LIN {X 0,Y 255.137,Z 1284.988,A -85,B 0,C 180,E1 17189.999,E2 17189.999} C_VEL
LIN {X 0,Y 254.468,Z 1282.963,A -85,B 0,C 180,E1 17196.81,E2 17196.81} C_VEL
LIN {X 0,Y 254.384,Z 1277.292,A -85,B 0,C 180,E1 17203.725,E2 17203.725} C_VEL
LIN {X 0,Y 256.072,Z 1266.53,A -85,B 0,C 180,E1 17211.61,E2 17211.61} C_VEL
LIN {X 0,Y 262.116,Z 1248.09,A -85,B 0,C 180,E1 17220.546,E2 17220.546} C_VEL
LIN {X 0,Y 272.188,Z 1225.017,A -85,B 0,C 180,E1 17228.249,E2 17228.249} C_VEL
LIN {X 0,Y 284.902,Z 1198.098,A -85,B 0,C 180,E1 17234.56,E2 17234.56} C_VEL
LIN {X 0,Y 299.3,Z 1166.688,A -85,B 0,C 180,E1 17239.69,E2 17239.69} C_VEL
LIN {X 0,Y 313.161,Z 1132.639,A -85,B 0,C 180,E1 17243.514,E2 17243.514} C_VEL
LIN {X 0,Y 320.37,Z 1111.086,A -85,B 0,C 180,E1 17245.369,E2 17245.369} C_VEL
LIN {X 0,Y 312.607,Z 1086.253,A -85,B 0,C 180,E1 17250.782,E2 17250.782} C_VEL
LIN {X 0,Y 302.724,Z 1063.673,A -85,B 0,C 180,E1 17257.275,E2 17257.275} C_VEL
LIN {X 0,Y 294.391,Z 1048.168,A -85,B 0,C 180,E1 17263.626,E2 17263.626} C_VEL
LIN {X 0,Y 291.709,Z 1044.139,A -85,B 0,C 180,E1 17266.011,E2 17266.011} C_VEL
LIN {X 0,Y 289.339,Z 1043.796,A -85,B 0,C 180,E1 17267.674,E2 17267.674} C_VEL
LIN {X 0,Y 285.403,Z 1045.605,A -85,B 0,C 180,E1 17270.235,E2 17270.235} C_VEL
LIN {X 0,Y 285.166,Z 1045.322,A -85,B 0,C 180,E1 17270.526,E2 17270.526} C_VEL
LIN {X 0,Y 284.224,Z 1042.423,A -85,B 0,C 180,E1 17272.373,E2 17272.373} C_VEL
LIN {X 0,Y 280.854,Z 1038.34,A -85,B 0,C 180,E1 17280,E2 17280} C_VEL
LIN {X 0,Y 280.283,Z 1039.511,A -85,B 0,C 180,E1 17286.181,E2 17286.181} C_VEL
LIN {X 0,Y 281.282,Z 1041.764,A -85,B 0,C 180,E1 17290.897,E2 17290.897} C_VEL
LIN {X 0,Y 284.187,Z 1051.363,A -85,B 0,C 180,E1 17298.577,E2 17298.577} C_VEL
LIN {X 0,Y 287.728,Z 1062.486,A -85,B 0,C 180,E1 17304.806,E2 17304.806} C_VEL
LIN {X 0,Y 291.72,Z 1079.881,A -85,B 0,C 180,E1 17312.089,E2 17312.089} C_VEL
LIN {X 0,Y 294.002,Z 1097.791,A -85,B 0,C 180,E1 17318.393,E2 17318.393} C_VEL
LIN {X 0,Y 294.147,Z 1115.354,A -85,B 0,C 180,E1 17324.094,E2 17324.094} C_VEL
LIN {X 0,Y 280.403,Z 1140.437,A -85,B 0,C 180,E1 17329.776,E2 17329.776} C_VEL
LIN {X 0,Y 267.571,Z 1161.591,A -85,B 0,C 180,E1 17336.74,E2 17336.74} C_VEL
LIN {X 0,Y 257.328,Z 1177.923,A -85,B 0,C 180,E1 17344.841,E2 17344.841} C_VEL
LIN {X 0,Y 251.436,Z 1187.855,A -85,B 0,C 180,E1 17352.539,E2 17352.539} C_VEL
LIN {X 0,Y 248.589,Z 1193.315,A -85,B 0,C 180,E1 17359.509,E2 17359.509} C_VEL
LIN {X 0,Y 247.507,Z 1195.971,A -85,B 0,C 180,E1 17366.506,E2 17366.506} C_VEL
LIN {X 0,Y 247.516,Z 1195.938,A -85,B 0,C 180,E1 17373.497,E2 17373.497} C_VEL
LIN {X 0,Y 249.137,Z 1192.204,A -85,B 0,C 180,E1 17382.24,E2 17382.24} C_VEL
LIN {X 0,Y 254.389,Z 1182.789,A -85,B 0,C 180,E1 17391.718,E2 17391.718} C_VEL
LIN {X 0,Y 263.096,Z 1168.574,A -85,B 0,C 180,E1 17400.125,E2 17400.125} C_VEL
LIN {X 0,Y 275.237,Z 1149.075,A -85,B 0,C 180,E1 17407.586,E2 17407.586} C_VEL
LIN {X 0,Y 288.938,Z 1125.242,A -85,B 0,C 180,E1 17413.775,E2 17413.775} C_VEL
LIN {X 0,Y 294.085,Z 1114.963,A -85,B 0,C 180,E1 17415.921,E2 17415.921} C_VEL
LIN {X 0,Y 293.829,Z 1096.412,A -85,B 0,C 180,E1 17421.957,E2 17421.957} C_VEL
LIN {X 0,Y 291.448,Z 1078.298,A -85,B 0,C 180,E1 17428.357,E2 17428.357} C_VEL
LIN {X 0,Y 287.609,Z 1062.12,A -85,B 0,C 180,E1 17435.183,E2 17435.183} C_VEL
LIN {X 0,Y 283.183,Z 1048.498,A -85,B 0,C 180,E1 17443.118,E2 17443.118} C_VEL
LIN {X 0,Y 280.59,Z 1040.614,A -85,B 0,C 180,E1 17450.716,E2 17450.716} C_VEL
LIN {X 0,Y 280.229,Z 1037.979,A -85,B 0,C 180,E1 17456.913,E2 17456.913} C_VEL
LIN {X 0,Y 280.753,Z 1037.906,A -85,B 0,C 180,E1 17460,E2 17460} C_VEL
LIN {X 0,Y 284.152,Z 1041.989,A -85,B 0,C 180,E1 17467.629,E2 17467.629} C_VEL
LIN {X 0,Y 290.868,Z 1054.58,A -85,B 0,C 180,E1 17475.805,E2 17475.805} C_VEL
LIN {X 0,Y 299.294,Z 1071.309,A -85,B 0,C 180,E1 17482.717,E2 17482.717} C_VEL
LIN {X 0,Y 307.569,Z 1091.151,A -85,B 0,C 180,E1 17488.576,E2 17488.576} C_VEL
LIN {X 0,Y 314.317,Z 1114.372,A -85,B 0,C 180,E1 17493.824,E2 17493.824} C_VEL
LIN {X 0,Y 300.167,Z 1151.228,A -85,B 0,C 180,E1 17497.349,E2 17497.349} C_VEL
LIN {X 0,Y 285.171,Z 1183.85,A -85,B 0,C 180,E1 17501.908,E2 17501.908} C_VEL
LIN {X 0,Y 270.591,Z 1213.505,A -85,B 0,C 180,E1 17507.992,E2 17507.992} C_VEL
LIN {X 0,Y 258.739,Z 1238.273,A -85,B 0,C 180,E1 17515.343,E2 17515.343} C_VEL
LIN {X 0,Y 250.401,Z 1258.673,A -85,B 0,C 180,E1 17524.093,E2 17524.093} C_VEL
LIN {X 0,Y 246.852,Z 1272.762,A -85,B 0,C 180,E1 17533.119,E2 17533.119} C_VEL
LIN {X 0,Y 246.557,Z 1280.502,A -85,B 0,C 180,E1 17541.197,E2 17541.197} C_VEL
LIN {X 0,Y 246.904,Z 1283.038,A -85,B 0,C 180,E1 17546.495,E2 17546.495} C_VEL
LIN {X 0,Y 247.367,Z 1283.617,A -85,B 0,C 180,E1 17549.999,E2 17549.999} C_VEL
LIN {X 0,Y 246.653,Z 1281.574,A -85,B 0,C 180,E1 17557.027,E2 17557.027} C_VEL
LIN {X 0,Y 246.583,Z 1275.874,A -85,B 0,C 180,E1 17564.168,E2 17564.168} C_VEL
LIN {X 0,Y 248.469,Z 1265.084,A -85,B 0,C 180,E1 17572.306,E2 17572.306} C_VEL
LIN {X 0,Y 254.378,Z 1248.105,A -85,B 0,C 180,E1 17580.899,E2 17580.899} C_VEL
LIN {X 0,Y 264.784,Z 1225.469,A -85,B 0,C 180,E1 17588.82,E2 17588.82} C_VEL
LIN {X 0,Y 278.173,Z 1198.463,A -85,B 0,C 180,E1 17595.396,E2 17595.396} C_VEL
LIN {X 0,Y 293.472,Z 1166.431,A -85,B 0,C 180,E1 17600.758,E2 17600.758} C_VEL
LIN {X 0,Y 307.806,Z 1132.751,A -85,B 0,C 180,E1 17604.588,E2 17604.588} C_VEL
LIN {X 0,Y 314.425,Z 1114.35,A -85,B 0,C 180,E1 17606.188,E2 17606.188} C_VEL
LIN {X 0,Y 307.121,Z 1089.98,A -85,B 0,C 180,E1 17611.779,E2 17611.779} C_VEL
LIN {X 0,Y 298.39,Z 1069.256,A -85,B 0,C 180,E1 17618.051,E2 17618.051} C_VEL
LIN {X 0,Y 290.985,Z 1054.781,A -85,B 0,C 180,E1 17624.202,E2 17624.202} C_VEL
LIN {X 0,Y 287.467,Z 1048.317,A -85,B 0,C 180,E1 17627.88,E2 17627.88} C_VEL
LIN {X 0,Y 285.166,Z 1045.322,A -85,B 0,C 180,E1 17630.526,E2 17630.526} C_VEL
LIN {X 0,Y 282.691,Z 1044.878,A -85,B 0,C 180,E1 17633.12,E2 17633.12} C_VEL
LIN {X 0,Y 278.853,Z 1047.015,A -85,B 0,C 180,E1 17637.566,E2 17637.566} C_VEL
LIN {X 0,Y 277.646,Z 1045.811,A -85,B 0,C 180,E1 17643.115,E2 17643.115} C_VEL
LIN {X 0,Y 278.291,Z 1049.367,A -85,B 0,C 180,E1 17651.015,E2 17651.015} C_VEL
LIN {X 0,Y 280.713,Z 1058.959,A -85,B 0,C 180,E1 17658.816,E2 17658.816} C_VEL
LIN {X 0,Y 284.069,Z 1071.905,A -85,B 0,C 180,E1 17665.873,E2 17665.873} C_VEL
LIN {X 0,Y 286.988,Z 1088.241,A -85,B 0,C 180,E1 17672.725,E2 17672.725} C_VEL
LIN {X 0,Y 288.302,Z 1105.417,A -85,B 0,C 180,E1 17678.908,E2 17678.908} C_VEL
LIN {X 0,Y 287.43,Z 1119.484,A -85,B 0,C 180,E1 17683.545,E2 17683.545} C_VEL
LIN {X 0,Y 272.089,Z 1145.854,A -85,B 0,C 180,E1 17689.856,E2 17689.856} C_VEL
LIN {X 0,Y 258.657,Z 1166.631,A -85,B 0,C 180,E1 17697.342,E2 17697.342} C_VEL
LIN {X 0,Y 248.492,Z 1182.013,A -85,B 0,C 180,E1 17705.895,E2 17705.895} C_VEL
LIN {X 0,Y 242.157,Z 1192.333,A -85,B 0,C 180,E1 17715.567,E2 17715.567} C_VEL
LIN {X 0,Y 240.061,Z 1196.366,A -85,B 0,C 180,E1 17722.779,E2 17722.779} C_VEL
LIN {X 0,Y 239.805,Z 1197.644,A -85,B 0,C 180,E1 17730.001,E2 17730.001} C_VEL
LIN {X 0,Y 240.054,Z 1196.316,A -85,B 0,C 180,E1 17737.224,E2 17737.224} C_VEL
LIN {X 0,Y 242.888,Z 1191.132,A -85,B 0,C 180,E1 17745.877,E2 17745.877} C_VEL
LIN {X 0,Y 249.513,Z 1180.492,A -85,B 0,C 180,E1 17755.047,E2 17755.047} C_VEL
LIN {X 0,Y 259.981,Z 1164.513,A -85,B 0,C 180,E1 17763.465,E2 17763.465} C_VEL
LIN {X 0,Y 273.017,Z 1144.178,A -85,B 0,C 180,E1 17770.501,E2 17770.501} C_VEL
LIN {X 0,Y 287.455,Z 1119.187,A -85,B 0,C 180,E1 17776.414,E2 17776.414} C_VEL
LIN {X 0,Y 288.073,Z 1103.066,A -85,B 0,C 180,E1 17781.791,E2 17781.791} C_VEL
LIN {X 0,Y 286.553,Z 1085.286,A -85,B 0,C 180,E1 17788.225,E2 17788.225} C_VEL
LIN {X 0,Y 283.263,Z 1068.551,A -85,B 0,C 180,E1 17795.523,E2 17795.523} C_VEL
LIN {X 0,Y 279.675,Z 1055.247,A -85,B 0,C 180,E1 17803.552,E2 17803.552} C_VEL
LIN {X 0,Y 277.738,Z 1048.039,A -85,B 0,C 180,E1 17810.62,E2 17810.62} C_VEL
LIN {X 0,Y 277.527,Z 1045.448,A -85,B 0,C 180,E1 17816.883,E2 17816.883} C_VEL
LIN {X 0,Y 278.18,Z 1045.394,A -85,B 0,C 180,E1 17820,E2 17820} C_VEL
LIN {X 0,Y 281.517,Z 1049.856,A -85,B 0,C 180,E1 17827.701,E2 17827.701} C_VEL
LIN {X 0,Y 287.342,Z 1061.146,A -85,B 0,C 180,E1 17835.223,E2 17835.223} C_VEL
LIN {X 0,Y 295.025,Z 1076.971,A -85,B 0,C 180,E1 17842.018,E2 17842.018} C_VEL
LIN {X 0,Y 302.864,Z 1097.215,A -85,B 0,C 180,E1 17848.183,E2 17848.183} C_VEL
LIN {X 0,Y 308.379,Z 1117.716,A -85,B 0,C 180,E1 17853.017,E2 17853.017} C_VEL
LIN {X 0,Y 294.309,Z 1151.941,A -85,B 0,C 180,E1 17856.342,E2 17856.342} C_VEL
LIN {X 0,Y 278.69,Z 1184.433,A -85,B 0,C 180,E1 17861.002,E2 17861.002} C_VEL
LIN {X 0,Y 263.917,Z 1213.139,A -85,B 0,C 180,E1 17867.067,E2 17867.067} C_VEL
LIN {X 0,Y 251.35,Z 1237.996,A -85,B 0,C 180,E1 17874.7,E2 17874.7} C_VEL
LIN {X 0,Y 243.009,Z 1257.212,A -85,B 0,C 180,E1 17883.242,E2 17883.242} C_VEL
LIN {X 0,Y 239.101,Z 1271.33,A -85,B 0,C 180,E1 17892.554,E2 17892.554} C_VEL
LIN {X 0,Y 238.711,Z 1279.1,A -85,B 0,C 180,E1 17900.906,E2 17900.906} C_VEL
LIN {X 0,Y 239.099,Z 1281.658,A -85,B 0,C 180,E1 17906.38,E2 17906.38} C_VEL
LIN {X 0,Y 239.571,Z 1282.241,A -85,B 0,C 180,E1 17909.999,E2 17909.999} C_VEL
LIN {X 0,Y 238.828,Z 1280.182,A -85,B 0,C 180,E1 17917.258,E2 17917.258} C_VEL
LIN {X 0,Y 238.788,Z 1274.454,A -85,B 0,C 180,E1 17924.641,E2 17924.641} C_VEL
LIN {X 0,Y 241.327,Z 1262.214,A -85,B 0,C 180,E1 17933.91,E2 17933.91} C_VEL
LIN {X 0,Y 248.706,Z 1243.691,A -85,B 0,C 180,E1 17943.096,E2 17943.096} C_VEL
LIN {X 0,Y 260.58,Z 1219.799,A -85,B 0,C 180,E1 17951.167,E2 17951.167} C_VEL
LIN {X 0,Y 275.272,Z 1191.427,A -85,B 0,C 180,E1 17957.735,E2 17957.735} C_VEL
LIN {X 0,Y 291.413,Z 1158.364,A -85,B 0,C 180,E1 17962.918,E2 17962.918} C_VEL
LIN {X 0,Y 306.908,Z 1121.702,A -85,B 0,C 180,E1 17966.704,E2 17966.704} C_VEL
LIN {X 0,Y 308.352,Z 1117.832,A -85,B 0,C 180,E1 17967.005,E2 17967.005} C_VEL
LIN {X 0,Y 302.38,Z 1095.769,A -85,B 0,C 180,E1 17972.257,E2 17972.257} C_VEL
LIN {X 0,Y 294.431,Z 1075.586,A -85,B 0,C 180,E1 17978.548,E2 17978.548} C_VEL
LIN {X 0,Y 287.451,Z 1061.347,A -85,B 0,C 180,E1 17984.783,E2 17984.783} C_VEL
LIN {X 0,Y 281.577,Z 1050.332,A -85,B 0,C 180,E1 17992.301,E2 17992.301} C_VEL
LIN {X 0,Y 278.853,Z 1047.015,A -85,B 0,C 180,E1 17997.566,E2 17997.566} C_VEL
LIN {X 0,Y 277.184,Z 1048.421,A -85,B 0,C 180,E1 18000.225,E2 18000.225} C_VEL
LIN {X 0,Y 274.51,Z 1053.721,A -85,B 0,C 180,E1 18004.671,E2 18004.671} C_VEL
LIN {X 0,Y 275.027,Z 1056.889,A -85,B 0,C 180,E1 18011.148,E2 18011.148} C_VEL
LIN {X 0,Y 277.086,Z 1066.535,A -85,B 0,C 180,E1 18019.071,E2 18019.071} C_VEL
LIN {X 0,Y 279.809,Z 1079.929,A -85,B 0,C 180,E1 18026.417,E2 18026.417} C_VEL
LIN {X 0,Y 281.865,Z 1096.426,A -85,B 0,C 180,E1 18033.396,E2 18033.396} C_VEL
LIN {X 0,Y 282.223,Z 1115.213,A -85,B 0,C 180,E1 18040.301,E2 18040.301} C_VEL
LIN {X 0,Y 281.309,Z 1122.317,A -85,B 0,C 180,E1 18042.676,E2 18042.676} C_VEL
LIN {X 0,Y 265.31,Z 1148.466,A -85,B 0,C 180,E1 18049.151,E2 18049.151} C_VEL
LIN {X 0,Y 252.074,Z 1168.017,A -85,B 0,C 180,E1 18056.377,E2 18056.377} C_VEL
LIN {X 0,Y 241.347,Z 1183.397,A -85,B 0,C 180,E1 18065.134,E2 18065.134} C_VEL
LIN {X 0,Y 234.584,Z 1193.714,A -85,B 0,C 180,E1 18075.091,E2 18075.091} C_VEL
LIN {X 0,Y 232.329,Z 1197.741,A -85,B 0,C 180,E1 18082.537,E2 18082.537} C_VEL
LIN {X 0,Y 232.043,Z 1199.014,A -85,B 0,C 180,E1 18090.001,E2 18090.001} C_VEL
LIN {X 0,Y 232.32,Z 1197.693,A -85,B 0,C 180,E1 18097.466,E2 18097.466} C_VEL
LIN {X 0,Y 235.525,Z 1192.196,A -85,B 0,C 180,E1 18106.757,E2 18106.757} C_VEL
LIN {X 0,Y 242.427,Z 1181.878,A -85,B 0,C 180,E1 18115.833,E2 18115.833} C_VEL
LIN {X 0,Y 253.473,Z 1165.899,A -85,B 0,C 180,E1 18124.443,E2 18124.443} C_VEL
LIN {X 0,Y 267.117,Z 1145.561,A -85,B 0,C 180,E1 18131.591,E2 18131.591} C_VEL
LIN {X 0,Y 281.614,Z 1120.703,A -85,B 0,C 180,E1 18137.677,E2 18137.677} C_VEL
LIN {X 0,Y 282.138,Z 1101.835,A -85,B 0,C 180,E1 18144.395,E2 18144.395} C_VEL
LIN {X 0,Y 280.573,Z 1085.149,A -85,B 0,C 180,E1 18151.051,E2 18151.051} C_VEL
LIN {X 0,Y 277.834,Z 1070.385,A -85,B 0,C 180,E1 18158.361,E2 18158.361} C_VEL
LIN {X 0,Y 275.38,Z 1059.996,A -85,B 0,C 180,E1 18165.725,E2 18165.725} C_VEL
LIN {X 0,Y 274.363,Z 1054.762,A -85,B 0,C 180,E1 18171.902,E2 18171.902} C_VEL
LIN {X 0,Y 275.302,Z 1052.79,A -85,B 0,C 180,E1 18180,E2 18180} C_VEL
LIN {X 0,Y 278.589,Z 1057.631,A -85,B 0,C 180,E1 18187.782,E2 18187.782} C_VEL
LIN {X 0,Y 284.37,Z 1069.061,A -85,B 0,C 180,E1 18195.386,E2 18195.386} C_VEL
LIN {X 0,Y 291.065,Z 1083.921,A -85,B 0,C 180,E1 18201.805,E2 18201.805} C_VEL
LIN {X 0,Y 298.159,Z 1103.61,A -85,B 0,C 180,E1 18207.913,E2 18207.913} C_VEL
LIN {X 0,Y 302.122,Z 1121.309,A -85,B 0,C 180,E1 18212.128,E2 18212.128} C_VEL
LIN {X 0,Y 286.317,Z 1157.309,A -85,B 0,C 180,E1 18215.852,E2 18215.852} C_VEL
LIN {X 0,Y 269.765,Z 1189.854,A -85,B 0,C 180,E1 18220.959,E2 18220.959} C_VEL
LIN {X 0,Y 254.209,Z 1218.36,A -85,B 0,C 180,E1 18227.613,E2 18227.613} C_VEL
LIN {X 0,Y 241.791,Z 1242.173,A -85,B 0,C 180,E1 18235.826,E2 18235.826} C_VEL
LIN {X 0,Y 233.939,Z 1260.374,A -85,B 0,C 180,E1 18245.048,E2 18245.048} C_VEL
LIN {X 0,Y 230.946,Z 1273.002,A -85,B 0,C 180,E1 18254.848,E2 18254.848} C_VEL
LIN {X 0,Y 231.033,Z 1278.783,A -85,B 0,C 180,E1 18262.493,E2 18262.493} C_VEL
LIN {X 0,Y 231.799,Z 1280.869,A -85,B 0,C 180,E1 18269.999,E2 18269.999} C_VEL
LIN {X 0,Y 231.004,Z 1278.791,A -85,B 0,C 180,E1 18277.506,E2 18277.506} C_VEL
LIN {X 0,Y 230.969,Z 1273.027,A -85,B 0,C 180,E1 18285.148,E2 18285.148} C_VEL
LIN {X 0,Y 233.955,Z 1260.411,A -85,B 0,C 180,E1 18294.947,E2 18294.947} C_VEL
LIN {X 0,Y 241.783,Z 1242.225,A -85,B 0,C 180,E1 18304.172,E2 18304.172} C_VEL
LIN {X 0,Y 254.331,Z 1218.322,A -85,B 0,C 180,E1 18312.41,E2 18312.41} C_VEL
LIN {X 0,Y 269.789,Z 1189.973,A -85,B 0,C 180,E1 18319.032,E2 18319.032} C_VEL
LIN {X 0,Y 286.198,Z 1157.626,A -85,B 0,C 180,E1 18324.132,E2 18324.132} C_VEL
LIN {X 0,Y 302.386,Z 1120.228,A -85,B 0,C 180,E1 18328.032,E2 18328.032} C_VEL
LIN {X 0,Y 296.511,Z 1098.509,A -85,B 0,C 180,E1 18333.558,E2 18333.558} C_VEL
LIN {X 0,Y 288.998,Z 1078.92,A -85,B 0,C 180,E1 18340.159,E2 18340.159} C_VEL
LIN {X 0,Y 282.367,Z 1065.494,A -85,B 0,C 180,E1 18346.873,E2 18346.873} C_VEL
LIN {X 0,Y 277.822,Z 1056.475,A -85,B 0,C 180,E1 18353.764,E2 18353.764} C_VEL
LIN {X 0,Y 275.395,Z 1053.192,A -85,B 0,C 180,E1 18360,E2 18360} C_VEL
LIN {X 0,Y 274.51,Z 1053.721,A -85,B 0,C 180,E1 18364.671,E2 18364.671} C_VEL
LIN {X 0,Y 273.488,Z 1056.922,A -85,B 0,C 180,E1 18367.32,E2 18367.32} C_VEL
LIN {X 0,Y 271.581,Z 1064.694,A -85,B 0,C 180,E1 18371.664,E2 18371.664} C_VEL
LIN {X 0,Y 273.152,Z 1074.035,A -85,B 0,C 180,E1 18379.357,E2 18379.357} C_VEL
LIN {X 0,Y 275.15,Z 1087.013,A -85,B 0,C 180,E1 18386.554,E2 18386.554} C_VEL
LIN {X 0,Y 276.433,Z 1104.04,A -85,B 0,C 180,E1 18393.918,E2 18393.918} C_VEL
LIN {X 0,Y 275.791,Z 1121.552,A -85,B 0,C 180,E1 18400.552,E2 18400.552} C_VEL
LIN {X 0,Y 274.354,Z 1126.477,A -85,B 0,C 180,E1 18402.065,E2 18402.065} C_VEL
LIN {X 0,Y 258.578,Z 1151.073,A -85,B 0,C 180,E1 18408.409,E2 18408.409} C_VEL
LIN {X 0,Y 244.227,Z 1171.179,A -85,B 0,C 180,E1 18416.216,E2 18416.216} C_VEL
LIN {X 0,Y 234.116,Z 1184.962,A -85,B 0,C 180,E1 18424.467,E2 18424.467} C_VEL
LIN {X 0,Y 227.041,Z 1195.093,A -85,B 0,C 180,E1 18434.583,E2 18434.583} C_VEL
LIN {X 0,Y 224.609,Z 1199.115,A -85,B 0,C 180,E1 18442.279,E2 18442.279} C_VEL
LIN {X 0,Y 224.263,Z 1200.387,A -85,B 0,C 180,E1 18450.001,E2 18450.001} C_VEL
LIN {X 0,Y 224.6,Z 1199.067,A -85,B 0,C 180,E1 18457.724,E2 18457.724} C_VEL
LIN {X 0,Y 228.04,Z 1193.576,A -85,B 0,C 180,E1 18467.326,E2 18467.326} C_VEL
LIN {X 0,Y 235.395,Z 1183.263,A -85,B 0,C 180,E1 18476.664,E2 18476.664} C_VEL
LIN {X 0,Y 247.049,Z 1167.284,A -85,B 0,C 180,E1 18485.471,E2 18485.471} C_VEL
LIN {X 0,Y 261.316,Z 1146.944,A -85,B 0,C 180,E1 18492.73,E2 18492.73} C_VEL
LIN {X 0,Y 275.285,Z 1124.783,A -85,B 0,C 180,E1 18498.19,E2 18498.19} C_VEL
LIN {X 0,Y 276.431,Z 1107.448,A -85,B 0,C 180,E1 18504.624,E2 18504.624} C_VEL
LIN {X 0,Y 275.643,Z 1091.63,A -85,B 0,C 180,E1 18511.157,E2 18511.157} C_VEL
LIN {X 0,Y 273.726,Z 1077.748,A -85,B 0,C 180,E1 18518.156,E2 18518.156} C_VEL
LIN {X 0,Y 271.83,Z 1067.361,A -85,B 0,C 180,E1 18525.535,E2 18525.535} C_VEL
LIN {X 0,Y 271.311,Z 1062.741,A -85,B 0,C 180,E1 18530.395,E2 18530.395} C_VEL
LIN {X 0,Y 271.765,Z 1060.081,A -85,B 0,C 180,E1 18538.175,E2 18538.175} C_VEL
LIN {X 0,Y 273.117,Z 1061.867,A -85,B 0,C 180,E1 18543.167,E2 18543.167} C_VEL
LIN {X 0,Y 275.552,Z 1065.297,A -85,B 0,C 180,E1 18547.869,E2 18547.869} C_VEL
LIN {X 0,Y 280.473,Z 1075.379,A -85,B 0,C 180,E1 18554.805,E2 18554.805} C_VEL
LIN {X 0,Y 286.994,Z 1090.804,A -85,B 0,C 180,E1 18561.595,E2 18561.595} C_VEL
LIN {X 0,Y 293.218,Z 1109.68,A -85,B 0,C 180,E1 18567.591,E2 18567.591} C_VEL
LIN {X 0,Y 296.304,Z 1123.552,A -85,B 0,C 180,E1 18571.117,E2 18571.117} C_VEL
LIN {X 0,Y 280.399,Z 1158.219,A -85,B 0,C 180,E1 18574.812,E2 18574.812} C_VEL
LIN {X 0,Y 264.396,Z 1188.386,A -85,B 0,C 180,E1 18579.599,E2 18579.599} C_VEL
LIN {X 0,Y 248.225,Z 1216.661,A -85,B 0,C 180,E1 18586.246,E2 18586.246} C_VEL
LIN {X 0,Y 234.908,Z 1240.693,A -85,B 0,C 180,E1 18594.678,E2 18594.678} C_VEL
LIN {X 0,Y 226.39,Z 1259.205,A -85,B 0,C 180,E1 18604.353,E2 18604.353} C_VEL
LIN {X 0,Y 223.163,Z 1271.576,A -85,B 0,C 180,E1 18614.306,E2 18614.306} C_VEL
LIN {X 0,Y 223.184,Z 1277.385,A -85,B 0,C 180,E1 18622.227,E2 18622.227} C_VEL
LIN {X 0,Y 224.004,Z 1279.494,A -85,B 0,C 180,E1 18629.999,E2 18629.999} C_VEL
LIN {X 0,Y 223.153,Z 1277.393,A -85,B 0,C 180,E1 18637.771,E2 18637.771} C_VEL
LIN {X 0,Y 223.44,Z 1269.868,A -85,B 0,C 180,E1 18647.48,E2 18647.48} C_VEL
LIN {X 0,Y 227.613,Z 1256.069,A -85,B 0,C 180,E1 18657.649,E2 18657.649} C_VEL
LIN {X 0,Y 237.411,Z 1236.13,A -85,B 0,C 180,E1 18667.229,E2 18667.229} C_VEL
LIN {X 0,Y 251.74,Z 1210.753,A -85,B 0,C 180,E1 18675.386,E2 18675.386} C_VEL
LIN {X 0,Y 267.656,Z 1182.671,A -85,B 0,C 180,E1 18681.466,E2 18681.466} C_VEL
LIN {X 0,Y 284.393,Z 1150.164,A -85,B 0,C 180,E1 18686.215,E2 18686.215} C_VEL
LIN {X 0,Y 296.348,Z 1123.596,A -85,B 0,C 180,E1 18688.903,E2 18688.903} C_VEL
LIN {X 0,Y 291.398,Z 1103.386,A -85,B 0,C 180,E1 18694.298,E2 18694.298} C_VEL
LIN {X 0,Y 284.559,Z 1084.411,A -85,B 0,C 180,E1 18700.967,E2 18700.967} C_VEL
LIN {X 0,Y 278.135,Z 1070.556,A -85,B 0,C 180,E1 18708.261,E2 18708.261} C_VEL
LIN {X 0,Y 274.861,Z 1063.925,A -85,B 0,C 180,E1 18713.696,E2 18713.696} C_VEL
LIN {X 0,Y 272.368,Z 1060.505,A -85,B 0,C 180,E1 18720,E2 18720} C_VEL
LIN {X 0,Y 271.244,Z 1061.555,A -85,B 0,C 180,E1 18726.388,E2 18726.388} C_VEL
LIN {X 0,Y 271.581,Z 1064.694,A -85,B 0,C 180,E1 18731.664,E2 18731.664} C_VEL
LIN {X 0,Y 270.77,Z 1069.677,A -85,B 0,C 180,E1 18734.225,E2 18734.225} C_VEL
LIN {X 0,Y 268.802,Z 1079.659,A -85,B 0,C 180,E1 18738.406,E2 18738.406} C_VEL
LIN {X 0,Y 270.16,Z 1091.867,A -85,B 0,C 180,E1 18745.643,E2 18745.643} C_VEL
LIN {X 0,Y 270.795,Z 1107.938,A -85,B 0,C 180,E1 18752.969,E2 18752.969} C_VEL
LIN {X 0,Y 269.763,Z 1124.431,A -85,B 0,C 180,E1 18759.545,E2 18759.545} C_VEL
LIN {X 0,Y 268.2,Z 1129.4,A -85,B 0,C 180,E1 18761.166,E2 18761.166} C_VEL
LIN {X 0,Y 251.888,Z 1153.681,A -85,B 0,C 180,E1 18767.628,E2 18767.628} C_VEL
LIN {X 0,Y 237.743,Z 1172.562,A -85,B 0,C 180,E1 18775.164,E2 18775.164} C_VEL
LIN {X 0,Y 226.498,Z 1187.063,A -85,B 0,C 180,E1 18784.183,E2 18784.183} C_VEL
LIN {X 0,Y 219.326,Z 1196.724,A -85,B 0,C 180,E1 18794.405,E2 18794.405} C_VEL
LIN {X 0,Y 216.886,Z 1200.491,A -85,B 0,C 180,E1 18802.003,E2 18802.003} C_VEL
LIN {X 0,Y 216.5,Z 1201.757,A -85,B 0,C 180,E1 18810.001,E2 18810.001} C_VEL
LIN {X 0,Y 216.876,Z 1200.444,A -85,B 0,C 180,E1 18818.001,E2 18818.001} C_VEL
LIN {X 0,Y 220.593,Z 1194.956,A -85,B 0,C 180,E1 18827.93,E2 18827.93} C_VEL
LIN {X 0,Y 228.407,Z 1184.65,A -85,B 0,C 180,E1 18837.548,E2 18837.548} C_VEL
LIN {X 0,Y 240.71,Z 1168.669,A -85,B 0,C 180,E1 18846.554,E2 18846.554} C_VEL
LIN {X 0,Y 255.612,Z 1148.33,A -85,B 0,C 180,E1 18853.923,E2 18853.923} C_VEL
LIN {X 0,Y 268.911,Z 1128.12,A -85,B 0,C 180,E1 18858.995,E2 18858.995} C_VEL
LIN {X 0,Y 270.721,Z 1110.985,A -85,B 0,C 180,E1 18865.629,E2 18865.629} C_VEL
LIN {X 0,Y 270.401,Z 1096.305,A -85,B 0,C 180,E1 18872.026,E2 18872.026} C_VEL
LIN {X 0,Y 269.027,Z 1082.387,A -85,B 0,C 180,E1 18879.548,E2 18879.548} C_VEL
LIN {X 0,Y 267.828,Z 1073.013,A -85,B 0,C 180,E1 18886.976,E2 18886.976} C_VEL
LIN {X 0,Y 267.633,Z 1068.742,A -85,B 0,C 180,E1 18892.996,E2 18892.996} C_VEL
LIN {X 0,Y 269.091,Z 1067.35,A -85,B 0,C 180,E1 18900,E2 18900} C_VEL
LIN {X 0,Y 272.261,Z 1072.811,A -85,B 0,C 180,E1 18907.964,E2 18907.964} C_VEL
LIN {X 0,Y 276.872,Z 1082.542,A -85,B 0,C 180,E1 18914.68,E2 18914.68} C_VEL
LIN {X 0,Y 282.86,Z 1097.905,A -85,B 0,C 180,E1 18921.516,E2 18921.516} C_VEL
LIN {X 0,Y 288.421,Z 1116.605,A -85,B 0,C 180,E1 18927.526,E2 18927.526} C_VEL
LIN {X 0,Y 290.028,Z 1127.06,A -85,B 0,C 180,E1 18930.183,E2 18930.183} C_VEL
LIN {X 0,Y 273.255,Z 1161.673,A -85,B 0,C 180,E1 18934.068,E2 18934.068} C_VEL
LIN {X 0,Y 254.944,Z 1194.349,A -85,B 0,C 180,E1 18939.692,E2 18939.692} C_VEL
LIN {X 0,Y 238.123,Z 1222.253,A -85,B 0,C 180,E1 18947.058,E2 18947.058} C_VEL
LIN {X 0,Y 225.883,Z 1243.496,A -85,B 0,C 180,E1 18955.398,E2 18955.398} C_VEL
LIN {X 0,Y 217.818,Z 1260.695,A -85,B 0,C 180,E1 18965.437,E2 18965.437} C_VEL
LIN {X 0,Y 215.193,Z 1272.011,A -85,B 0,C 180,E1 18975.791,E2 18975.791} C_VEL
LIN {X 0,Y 215.341,Z 1275.988,A -85,B 0,C 180,E1 18981.942,E2 18981.942} C_VEL
LIN {X 0,Y 216.228,Z 1278.121,A -85,B 0,C 180,E1 18989.999,E2 18989.999} C_VEL
LIN {X 0,Y 215.31,Z 1275.996,A -85,B 0,C 180,E1 18998.056,E2 18998.056} C_VEL
LIN {X 0,Y 215.669,Z 1268.586,A -85,B 0,C 180,E1 19007.985,E2 19007.985} C_VEL
LIN {X 0,Y 220.329,Z 1254.613,A -85,B 0,C 180,E1 19018.646,E2 19018.646} C_VEL
LIN {X 0,Y 230.802,Z 1234.589,A -85,B 0,C 180,E1 19028.515,E2 19028.515} C_VEL
LIN {X 0,Y 245.971,Z 1209.298,A -85,B 0,C 180,E1 19036.761,E2 19036.761} C_VEL
LIN {X 0,Y 263.126,Z 1180.317,A -85,B 0,C 180,E1 19043.027,E2 19043.027} C_VEL
LIN {X 0,Y 279.929,Z 1148.726,A -85,B 0,C 180,E1 19047.606,E2 19047.606} C_VEL
LIN {X 0,Y 290.064,Z 1127.219,A -85,B 0,C 180,E1 19049.82,E2 19049.82} C_VEL
LIN {X 0,Y 286.832,Z 1110.583,A -85,B 0,C 180,E1 19054.277,E2 19054.277} C_VEL
LIN {X 0,Y 281.156,Z 1093.136,A -85,B 0,C 180,E1 19060.401,E2 19060.401} C_VEL
LIN {X 0,Y 275.365,Z 1079.469,A -85,B 0,C 180,E1 19067.338,E2 19067.338} C_VEL
LIN {X 0,Y 271.609,Z 1071.324,A -85,B 0,C 180,E1 19073.621,E2 19073.621} C_VEL
LIN {X 0,Y 269.168,Z 1067.741,A -85,B 0,C 180,E1 19080,E2 19080} C_VEL
LIN {X 0,Y 267.825,Z 1068.746,A -85,B 0,C 180,E1 19086.47,E2 19086.47} C_VEL
LIN {X 0,Y 267.991,Z 1071.566,A -85,B 0,C 180,E1 19091.366,E2 19091.366} C_VEL
LIN {X 0,Y 268.802,Z 1079.659,A -85,B 0,C 180,E1 19098.406,E2 19098.406} C_VEL
LIN {X 0,Y 267.908,Z 1085.537,A -85,B 0,C 180,E1 19100.905,E2 19100.905} C_VEL
LIN {X 0,Y 265.195,Z 1097.161,A -85,B 0,C 180,E1 19104.934,E2 19104.934} C_VEL
LIN {X 0,Y 265.169,Z 1112.859,A -85,B 0,C 180,E1 19112.435,E2 19112.435} C_VEL
LIN {X 0,Y 263.537,Z 1128.67,A -85,B 0,C 180,E1 19119.038,E2 19119.038} C_VEL
LIN {X 0,Y 261.606,Z 1133.119,A -85,B 0,C 180,E1 19120.404,E2 19120.404} C_VEL
LIN {X 0,Y 244.315,Z 1157.526,A -85,B 0,C 180,E1 19127.204,E2 19127.204} C_VEL
LIN {X 0,Y 229.038,Z 1176.864,A -85,B 0,C 180,E1 19135.548,E2 19135.548} C_VEL
LIN {X 0,Y 217.466,Z 1190.916,A -85,B 0,C 180,E1 19145.398,E2 19145.398} C_VEL
LIN {X 0,Y 210.852,Z 1199.456,A -85,B 0,C 180,E1 19156.074,E2 19156.074} C_VEL
LIN {X 0,Y 208.671,Z 1202.838,A -85,B 0,C 180,E1 19165.854,E2 19165.854} C_VEL
LIN {X 0,Y 208.691,Z 1202.806,A -85,B 0,C 180,E1 19174.148,E2 19174.148} C_VEL
LIN {X 0,Y 210.852,Z 1199.389,A -85,B 0,C 180,E1 19183.93,E2 19183.93} C_VEL
LIN {X 0,Y 217.543,Z 1190.785,A -85,B 0,C 180,E1 19194.596,E2 19194.596} C_VEL
LIN {X 0,Y 229.151,Z 1176.575,A -85,B 0,C 180,E1 19204.497,E2 19204.497} C_VEL
LIN {X 0,Y 244.44,Z 1157.232,A -85,B 0,C 180,E1 19212.773,E2 19212.773} C_VEL
LIN {X 0,Y 261.678,Z 1132.828,A -85,B 0,C 180,E1 19219.547,E2 19219.547} C_VEL
LIN {X 0,Y 263.587,Z 1127.513,A -85,B 0,C 180,E1 19221.343,E2 19221.343} C_VEL
LIN {X 0,Y 265.192,Z 1111.316,A -85,B 0,C 180,E1 19228.084,E2 19228.084} C_VEL
LIN {X 0,Y 265.085,Z 1097.51,A -85,B 0,C 180,E1 19234.729,E2 19234.729} C_VEL
LIN {X 0,Y 264.375,Z 1086.053,A -85,B 0,C 180,E1 19241.705,E2 19241.705} C_VEL
LIN {X 0,Y 264.013,Z 1077.189,A -85,B 0,C 180,E1 19250.127,E2 19250.127} C_VEL
LIN {X 0,Y 264.733,Z 1074.531,A -85,B 0,C 180,E1 19256.733,E2 19256.733} C_VEL
LIN {X 0,Y 265.661,Z 1074.475,A -85,B 0,C 180,E1 19260,E2 19260} C_VEL
LIN {X 0,Y 268.825,Z 1080.148,A -85,B 0,C 180,E1 19268.067,E2 19268.067} C_VEL
LIN {X 0,Y 273.451,Z 1090.735,A -85,B 0,C 180,E1 19275.196,E2 19275.196} C_VEL
LIN {X 0,Y 278.683,Z 1105.341,A -85,B 0,C 180,E1 19281.644,E2 19281.644} C_VEL
LIN {X 0,Y 283.453,Z 1124.436,A -85,B 0,C 180,E1 19287.763,E2 19287.763} C_VEL
LIN {X 0,Y 283.88,Z 1130.362,A -85,B 0,C 180,E1 19289.204,E2 19289.204} C_VEL
LIN {X 0,Y 266.211,Z 1164.813,A -85,B 0,C 180,E1 19293.267,E2 19293.267} C_VEL
LIN {X 0,Y 248.39,Z 1195.008,A -85,B 0,C 180,E1 19298.705,E2 19298.705} C_VEL
LIN {X 0,Y 232.061,Z 1220.81,A -85,B 0,C 180,E1 19305.665,E2 19305.665} C_VEL
LIN {X 0,Y 219.089,Z 1242.027,A -85,B 0,C 180,E1 19314.163,E2 19314.163} C_VEL
LIN {X 0,Y 210.36,Z 1259.242,A -85,B 0,C 180,E1 19324.505,E2 19324.505} C_VEL
LIN {X 0,Y 207.366,Z 1270.584,A -85,B 0,C 180,E1 19335.243,E2 19335.243} C_VEL
LIN {X 0,Y 207.491,Z 1274.588,A -85,B 0,C 180,E1 19341.635,E2 19341.635} C_VEL
LIN {X 0,Y 208.454,Z 1276.75,A -85,B 0,C 180,E1 19349.999,E2 19349.999} C_VEL
LIN {X 0,Y 207.462,Z 1274.597,A -85,B 0,C 180,E1 19358.363,E2 19358.363} C_VEL
LIN {X 0,Y 207.847,Z 1267.57,A -85,B 0,C 180,E1 19368.218,E2 19368.218} C_VEL
LIN {X 0,Y 213.089,Z 1253.151,A -85,B 0,C 180,E1 19379.715,E2 19379.715} C_VEL
LIN {X 0,Y 224.604,Z 1232.62,A -85,B 0,C 180,E1 19390.044,E2 19390.044} C_VEL
LIN {X 0,Y 240.338,Z 1207.83,A -85,B 0,C 180,E1 19398.209,E2 19398.209} C_VEL
LIN {X 0,Y 258.143,Z 1179.058,A -85,B 0,C 180,E1 19404.454,E2 19404.454} C_VEL
LIN {X 0,Y 275.684,Z 1147.265,A -85,B 0,C 180,E1 19409.033,E2 19409.033} C_VEL
LIN {X 0,Y 284.348,Z 1128.948,A -85,B 0,C 180,E1 19411.038,E2 19411.038} C_VEL
LIN {X 0,Y 279.924,Z 1109.595,A -85,B 0,C 180,E1 19416.919,E2 19416.919} C_VEL
LIN {X 0,Y 274.794,Z 1093.979,A -85,B 0,C 180,E1 19423.245,E2 19423.245} C_VEL
LIN {X 0,Y 269.752,Z 1082.391,A -85,B 0,C 180,E1 19430.339,E2 19430.339} C_VEL
LIN {X 0,Y 267.369,Z 1077.444,A -85,B 0,C 180,E1 19435.144,E2 19435.144} C_VEL
LIN {X 0,Y 265.71,Z 1074.87,A -85,B 0,C 180,E1 19440,E2 19440} C_VEL
LIN {X 0,Y 264.298,Z 1075.869,A -85,B 0,C 180,E1 19446.557,E2 19446.557} C_VEL
LIN {X 0,Y 264.1,Z 1078.768,A -85,B 0,C 180,E1 19451.535,E2 19451.535} C_VEL
LIN {X 0,Y 264.552,Z 1087.014,A -85,B 0,C 180,E1 19458.761,E2 19458.761} C_VEL
LIN {X 0,Y 265.195,Z 1097.161,A -85,B 0,C 180,E1 19464.934,E2 19464.934} C_VEL
LIN {X 0,Y 263.751,Z 1103.841,A -85,B 0,C 180,E1 19467.363,E2 19467.363} C_VEL
LIN {X 0,Y 259.553,Z 1116.359,A -85,B 0,C 180,E1 19471.275,E2 19471.275} C_VEL
LIN {X 0,Y 257.408,Z 1132.121,A -85,B 0,C 180,E1 19478.21,E2 19478.21} C_VEL
LIN {X 0,Y 254.862,Z 1137.119,A -85,B 0,C 180,E1 19479.673,E2 19479.673} C_VEL
LIN {X 0,Y 236.948,Z 1160.989,A -85,B 0,C 180,E1 19486.671,E2 19486.671} C_VEL
LIN {X 0,Y 221.681,Z 1179.271,A -85,B 0,C 180,E1 19495.009,E2 19495.009} C_VEL
LIN {X 0,Y 210.345,Z 1192.302,A -85,B 0,C 180,E1 19504.506,E2 19504.506} C_VEL
LIN {X 0,Y 203.809,Z 1200.142,A -85,B 0,C 180,E1 19514.255,E2 19514.255} C_VEL
LIN {X 0,Y 200.913,Z 1204.211,A -85,B 0,C 180,E1 19525.694,E2 19525.694} C_VEL
LIN {X 0,Y 200.931,Z 1204.179,A -85,B 0,C 180,E1 19534.309,E2 19534.309} C_VEL
LIN {X 0,Y 203.811,Z 1200.058,A -85,B 0,C 180,E1 19545.747,E2 19545.747} C_VEL
LIN {X 0,Y 211.483,Z 1190.953,A -85,B 0,C 180,E1 19556.577,E2 19556.577} C_VEL
LIN {X 0,Y 224.265,Z 1176.12,A -85,B 0,C 180,E1 19566.592,E2 19566.592} C_VEL
LIN {X 0,Y 240.63,Z 1156.163,A -85,B 0,C 180,E1 19574.871,E2 19574.871} C_VEL
LIN {X 0,Y 257.037,Z 1133.068,A -85,B 0,C 180,E1 19581.298,E2 19581.298} C_VEL
LIN {X 0,Y 259.475,Z 1116.612,A -85,B 0,C 180,E1 19588.441,E2 19588.441} C_VEL
LIN {X 0,Y 260.003,Z 1103.248,A -85,B 0,C 180,E1 19595.155,E2 19595.155} C_VEL
LIN {X 0,Y 259.934,Z 1092.637,A -85,B 0,C 180,E1 19601.88,E2 19601.88} C_VEL
LIN {X 0,Y 260.162,Z 1083.96,A -85,B 0,C 180,E1 19610.425,E2 19610.425} C_VEL
LIN {X 0,Y 261.071,Z 1081.579,A -85,B 0,C 180,E1 19616.687,E2 19616.687} C_VEL
LIN {X 0,Y 262.127,Z 1081.553,A -85,B 0,C 180,E1 19620,E2 19620} C_VEL
LIN {X 0,Y 265.247,Z 1087.41,A -85,B 0,C 180,E1 19628.176,E2 19628.176} C_VEL
LIN {X 0,Y 269.723,Z 1098.491,A -85,B 0,C 180,E1 19635.557,E2 19635.557} C_VEL
LIN {X 0,Y 274.589,Z 1113.882,A -85,B 0,C 180,E1 19642.197,E2 19642.197} C_VEL
LIN {X 0,Y 278.211,Z 1131.668,A -85,B 0,C 180,E1 19647.89,E2 19647.89} C_VEL
LIN {X 0,Y 260.508,Z 1165.559,A -85,B 0,C 180,E1 19652.093,E2 19652.093} C_VEL
LIN {X 0,Y 242.48,Z 1194.779,A -85,B 0,C 180,E1 19657.462,E2 19657.462} C_VEL
LIN {X 0,Y 225.785,Z 1219.844,A -85,B 0,C 180,E1 19664.357,E2 19664.357} C_VEL
LIN {X 0,Y 211.15,Z 1242.508,A -85,B 0,C 180,E1 19673.87,E2 19673.87} C_VEL
LIN {X 0,Y 202.349,Z 1259.135,A -85,B 0,C 180,E1 19684.607,E2 19684.607} C_VEL
LIN {X 0,Y 199.576,Z 1269.161,A -85,B 0,C 180,E1 19694.653,E2 19694.653} C_VEL
LIN {X 0,Y 199.64,Z 1273.186,A -85,B 0,C 180,E1 19701.304,E2 19701.304} C_VEL
LIN {X 0,Y 200.673,Z 1275.376,A -85,B 0,C 180,E1 19709.998,E2 19709.998} C_VEL
LIN {X 0,Y 199.611,Z 1273.196,A -85,B 0,C 180,E1 19718.695,E2 19718.695} C_VEL
LIN {X 0,Y 200.145,Z 1266.137,A -85,B 0,C 180,E1 19728.945,E2 19728.945} C_VEL
LIN {X 0,Y 205.934,Z 1251.69,A -85,B 0,C 180,E1 19740.858,E2 19740.858} C_VEL
LIN {X 0,Y 218.066,Z 1231.532,A -85,B 0,C 180,E1 19751.295,E2 19751.295} C_VEL
LIN {X 0,Y 234.865,Z 1206.361,A -85,B 0,C 180,E1 19759.725,E2 19759.725} C_VEL
LIN {X 0,Y 253.576,Z 1177.339,A -85,B 0,C 180,E1 19766.023,E2 19766.023} C_VEL
LIN {X 0,Y 271.894,Z 1145.274,A -85,B 0,C 180,E1 19770.565,E2 19770.565} C_VEL
LIN {X 0,Y 278.324,Z 1131.739,A -85,B 0,C 180,E1 19772.112,E2 19772.112} C_VEL
LIN {X 0,Y 274.35,Z 1112.995,A -85,B 0,C 180,E1 19778.208,E2 19778.208} C_VEL
LIN {X 0,Y 269.449,Z 1097.737,A -85,B 0,C 180,E1 19784.957,E2 19784.957} C_VEL
LIN {X 0,Y 265.31,Z 1087.716,A -85,B 0,C 180,E1 19791.826,E2 19791.826} C_VEL
LIN {X 0,Y 263.136,Z 1083.563,A -85,B 0,C 180,E1 19796.713,E2 19796.713} C_VEL
LIN {X 0,Y 262.165,Z 1081.934,A -85,B 0,C 180,E1 19800,E2 19800} C_VEL
LIN {X 0,Y 260.452,Z 1082.869,A -85,B 0,C 180,E1 19806.654,E2 19806.654} C_VEL
LIN {X 0,Y 260.107,Z 1085.885,A -85,B 0,C 180,E1 19811.715,E2 19811.715} C_VEL
LIN {X 0,Y 260.096,Z 1094.746,A -85,B 0,C 180,E1 19819.484,E2 19819.484} C_VEL
LIN {X 0,Y 260.009,Z 1107.606,A -85,B 0,C 180,E1 19826.979,E2 19826.979} C_VEL
LIN {X 0,Y 259.553,Z 1116.359,A -85,B 0,C 180,E1 19831.275,E2 19831.275} C_VEL
LIN {X 0,Y 257.033,Z 1123.592,A -85,B 0,C 180,E1 19833.661,E2 19833.661} C_VEL
LIN {X 0,Y 251.207,Z 1136.084,A -85,B 0,C 180,E1 19837.56,E2 19837.56} C_VEL
LIN {X 0,Y 234.068,Z 1159.051,A -85,B 0,C 180,E1 19844.177,E2 19844.177} C_VEL
LIN {X 0,Y 217.451,Z 1178.253,A -85,B 0,C 180,E1 19852.445,E2 19852.445} C_VEL
LIN {X 0,Y 204.573,Z 1192.302,A -85,B 0,C 180,E1 19862.267,E2 19862.267} C_VEL
LIN {X 0,Y 196.299,Z 1201.521,A -85,B 0,C 180,E1 19873.636,E2 19873.636} C_VEL
LIN {X 0,Y 193.147,Z 1205.585,A -85,B 0,C 180,E1 19885.521,E2 19885.521} C_VEL
LIN {X 0,Y 193.162,Z 1205.554,A -85,B 0,C 180,E1 19894.482,E2 19894.482} C_VEL
LIN {X 0,Y 196.303,Z 1201.437,A -85,B 0,C 180,E1 19906.366,E2 19906.366} C_VEL
LIN {X 0,Y 204.83,Z 1191.978,A -85,B 0,C 180,E1 19917.869,E2 19917.869} C_VEL
LIN {X 0,Y 217.594,Z 1177.981,A -85,B 0,C 180,E1 19927.572,E2 19927.572} C_VEL
LIN {X 0,Y 234.158,Z 1158.774,A -85,B 0,C 180,E1 19935.805,E2 19935.805} C_VEL
LIN {X 0,Y 250.803,Z 1137.023,A -85,B 0,C 180,E1 19941.946,E2 19941.946} C_VEL
LIN {X 0,Y 253.877,Z 1120.815,A -85,B 0,C 180,E1 19949.301,E2 19949.301} C_VEL
LIN {X 0,Y 254.992,Z 1107.171,A -85,B 0,C 180,E1 19956.632,E2 19956.632} C_VEL
LIN {X 0,Y 255.403,Z 1096.951,A -85,B 0,C 180,E1 19963.801,E2 19963.801} C_VEL
LIN {X 0,Y 255.925,Z 1091.307,A -85,B 0,C 180,E1 19969.812,E2 19969.812} C_VEL
LIN {X 0,Y 257.21,Z 1088.539,A -85,B 0,C 180,E1 19976.637,E2 19976.637} C_VEL
LIN {X 0,Y 258.292,Z 1088.467,A -85,B 0,C 180,E1 19980,E2 19980} C_VEL
LIN {X 0,Y 260.676,Z 1092.679,A -85,B 0,C 180,E1 19986.648,E2 19986.648} C_VEL
LIN {X 0,Y 264.059,Z 1101.363,A -85,B 0,C 180,E1 19993.213,E2 19993.213} C_VEL
LIN {X 0,Y 268.184,Z 1114.463,A -85,B 0,C 180,E1 19999.73,E2 19999.73} C_VEL
LIN {X 0,Y 271.912,Z 1131.735,A -85,B 0,C 180,E1 20005.946,E2 20005.946} C_VEL
LIN {X 0,Y 272.149,Z 1135.691,A -85,B 0,C 180,E1 20007.045,E2 20007.045} C_VEL
LIN {X 0,Y 252.288,Z 1170.652,A -85,B 0,C 180,E1 20011.531,E2 20011.531} C_VEL
LIN {X 0,Y 232.137,Z 1201.196,A -85,B 0,C 180,E1 20017.752,E2 20017.752} C_VEL
LIN {X 0,Y 214.135,Z 1226.759,A -85,B 0,C 180,E1 20025.9,E2 20025.9} C_VEL
LIN {X 0,Y 200.865,Z 1246.702,A -85,B 0,C 180,E1 20035.725,E2 20035.725} C_VEL
LIN {X 0,Y 193.415,Z 1261.541,A -85,B 0,C 180,E1 20047.038,E2 20047.038} C_VEL
LIN {X 0,Y 191.669,Z 1269.269,A -85,B 0,C 180,E1 20056.337,E2 20056.337} C_VEL
LIN {X 0,Y 192.148,Z 1273.351,A -85,B 0,C 180,E1 20065.494,E2 20065.494} C_VEL
LIN {X 0,Y 192.872,Z 1274,A -85,B 0,C 180,E1 20069.998,E2 20069.998} C_VEL
LIN {X 0,Y 191.779,Z 1271.798,A -85,B 0,C 180,E1 20079.053,E2 20079.053} C_VEL
LIN {X 0,Y 192.465,Z 1264.633,A -85,B 0,C 180,E1 20089.811,E2 20089.811} C_VEL
LIN {X 0,Y 198.859,Z 1250.227,A -85,B 0,C 180,E1 20102.084,E2 20102.084} C_VEL
LIN {X 0,Y 211.658,Z 1230.421,A -85,B 0,C 180,E1 20112.631,E2 20112.631} C_VEL
LIN {X 0,Y 229.596,Z 1204.901,A -85,B 0,C 180,E1 20121.302,E2 20121.302} C_VEL
LIN {X 0,Y 248.942,Z 1176.085,A -85,B 0,C 180,E1 20127.561,E2 20127.561} C_VEL
LIN {X 0,Y 267.919,Z 1143.941,A -85,B 0,C 180,E1 20132.074,E2 20132.074} C_VEL
LIN {X 0,Y 272.168,Z 1135.974,A -85,B 0,C 180,E1 20132.933,E2 20132.933} C_VEL
LIN {X 0,Y 269.826,Z 1120.915,A -85,B 0,C 180,E1 20137.822,E2 20137.822} C_VEL
LIN {X 0,Y 265.592,Z 1105.546,A -85,B 0,C 180,E1 20144.524,E2 20144.524} C_VEL
LIN {X 0,Y 261.423,Z 1094.826,A -85,B 0,C 180,E1 20151.703,E2 20151.703} C_VEL
LIN {X 0,Y 259.309,Z 1090.518,A -85,B 0,C 180,E1 20156.664,E2 20156.664} C_VEL
LIN {X 0,Y 258.317,Z 1088.859,A -85,B 0,C 180,E1 20160,E2 20160} C_VEL
LIN {X 0,Y 256.505,Z 1089.808,A -85,B 0,C 180,E1 20166.757,E2 20166.757} C_VEL
LIN {X 0,Y 255.873,Z 1092.903,A -85,B 0,C 180,E1 20171.912,E2 20171.912} C_VEL
LIN {X 0,Y 255.363,Z 1101.983,A -85,B 0,C 180,E1 20179.863,E2 20179.863} C_VEL
LIN {X 0,Y 254.568,Z 1114.394,A -85,B 0,C 180,E1 20187.235,E2 20187.235} C_VEL
LIN {X 0,Y 252.696,Z 1128.866,A -85,B 0,C 180,E1 20194.304,E2 20194.304} C_VEL
LIN {X 0,Y 251.207,Z 1136.084,A -85,B 0,C 180,E1 20197.56,E2 20197.56} C_VEL
LIN {X 0,Y 248.162,Z 1141.033,A -85,B 0,C 180,E1 20198.946,E2 20198.946} C_VEL
LIN {X 0,Y 231.877,Z 1156.726,A -85,B 0,C 180,E1 20201.542,E2 20201.542} C_VEL
LIN {X 0,Y 230.734,Z 1157.967,A -85,B 0,C 180,E1 20201.925,E2 20201.925} C_VEL
LIN {X 0,Y 212.711,Z 1178.101,A -85,B 0,C 180,E1 20210.324,E2 20210.324} C_VEL
LIN {X 0,Y 199.253,Z 1192.042,A -85,B 0,C 180,E1 20219.739,E2 20219.739} C_VEL
LIN {X 0,Y 189.626,Z 1201.991,A -85,B 0,C 180,E1 20231.441,E2 20231.441} C_VEL
LIN {X 0,Y 186.033,Z 1205.997,A -85,B 0,C 180,E1 20240.665,E2 20240.665} C_VEL
LIN {X 0,Y 185.432,Z 1207.239,A -85,B 0,C 180,E1 20250.002,E2 20250.002} C_VEL
LIN {X 0,Y 186.021,Z 1205.953,A -85,B 0,C 180,E1 20259.339,E2 20259.339} C_VEL
LIN {X 0,Y 191.047,Z 1200.484,A -85,B 0,C 180,E1 20270.822,E2 20270.822} C_VEL
LIN {X 0,Y 201.093,Z 1190.196,A -85,B 0,C 180,E1 20281.689,E2 20281.689} C_VEL
LIN {X 0,Y 216.291,Z 1174.218,A -85,B 0,C 180,E1 20291.515,E2 20291.515} C_VEL
LIN {X 0,Y 234.052,Z 1153.869,A -85,B 0,C 180,E1 20299.252,E2 20299.252} C_VEL
LIN {X 0,Y 244.991,Z 1139.618,A -85,B 0,C 180,E1 20303.202,E2 20303.202} C_VEL
LIN {X 0,Y 248.341,Z 1124.861,A -85,B 0,C 180,E1 20310.289,E2 20310.289} C_VEL
LIN {X 0,Y 249.97,Z 1111.705,A -85,B 0,C 180,E1 20317.794,E2 20317.794} C_VEL
LIN {X 0,Y 250.867,Z 1103.115,A -85,B 0,C 180,E1 20324.249,E2 20324.249} C_VEL
LIN {X 0,Y 251.621,Z 1098.241,A -85,B 0,C 180,E1 20329.636,E2 20329.636} C_VEL
LIN {X 0,Y 253.128,Z 1095.373,A -85,B 0,C 180,E1 20336.583,E2 20336.583} C_VEL
LIN {X 0,Y 254.347,Z 1095.338,A -85,B 0,C 180,E1 20340,E2 20340} C_VEL
LIN {X 0,Y 256.727,Z 1099.708,A -85,B 0,C 180,E1 20346.751,E2 20346.751} C_VEL
LIN {X 0,Y 259.874,Z 1108.586,A -85,B 0,C 180,E1 20353.43,E2 20353.43} C_VEL
LIN {X 0,Y 263.662,Z 1122.112,A -85,B 0,C 180,E1 20360.083,E2 20360.083} C_VEL
LIN {X 0,Y 266.356,Z 1137.281,A -85,B 0,C 180,E1 20365.61,E2 20365.61} C_VEL
LIN {X 0,Y 262.453,Z 1145.347,A -85,B 0,C 180,E1 20366.68,E2 20366.68} C_VEL
LIN {X 0,Y 241.576,Z 1179.031,A -85,B 0,C 180,E1 20371.58,E2 20371.58} C_VEL
LIN {X 0,Y 221.059,Z 1208.061,A -85,B 0,C 180,E1 20378.367,E2 20378.367} C_VEL
LIN {X 0,Y 203.131,Z 1232.245,A -85,B 0,C 180,E1 20387.32,E2 20387.32} C_VEL
LIN {X 0,Y 190.91,Z 1250.309,A -85,B 0,C 180,E1 20397.753,E2 20397.753} C_VEL
LIN {X 0,Y 184.772,Z 1263.187,A -85,B 0,C 180,E1 20409.355,E2 20409.355} C_VEL
LIN {X 0,Y 183.96,Z 1270.383,A -85,B 0,C 180,E1 20420.556,E2 20420.556} C_VEL
LIN {X 0,Y 185.085,Z 1272.626,A -85,B 0,C 180,E1 20429.998,E2 20429.998} C_VEL
LIN {X 0,Y 183.902,Z 1270.108,A -85,B 0,C 180,E1 20440.062,E2 20440.062} C_VEL
LIN {X 0,Y 184.793,Z 1263.191,A -85,B 0,C 180,E1 20450.67,E2 20450.67} C_VEL
LIN {X 0,Y 191.859,Z 1248.76,A -85,B 0,C 180,E1 20463.404,E2 20463.404} C_VEL
LIN {X 0,Y 205.612,Z 1228.954,A -85,B 0,C 180,E1 20474.202,E2 20474.202} C_VEL
LIN {X 0,Y 224.283,Z 1203.711,A -85,B 0,C 180,E1 20482.888,E2 20482.888} C_VEL
LIN {X 0,Y 244.713,Z 1174.494,A -85,B 0,C 180,E1 20489.214,E2 20489.214} C_VEL
LIN {X 0,Y 263.912,Z 1143.019,A -85,B 0,C 180,E1 20493.581,E2 20493.581} C_VEL
LIN {X 0,Y 266.406,Z 1137.451,A -85,B 0,C 180,E1 20494.385,E2 20494.385} C_VEL
LIN {X 0,Y 263.29,Z 1120.3,A -85,B 0,C 180,E1 20500.759,E2 20500.759} C_VEL
LIN {X 0,Y 259.521,Z 1107.415,A -85,B 0,C 180,E1 20507.406,E2 20507.406} C_VEL
LIN {X 0,Y 256.101,Z 1098.487,A -85,B 0,C 180,E1 20514.93,E2 20514.93} C_VEL
LIN {X 0,Y 254.361,Z 1095.705,A -85,B 0,C 180,E1 20520,E2 20520} C_VEL
LIN {X 0,Y 252.321,Z 1096.646,A -85,B 0,C 180,E1 20526.869,E2 20526.869} C_VEL
LIN {X 0,Y 251.355,Z 1100.242,A -85,B 0,C 180,E1 20532.642,E2 20532.642} C_VEL
LIN {X 0,Y 250.361,Z 1109.169,A -85,B 0,C 180,E1 20540.332,E2 20540.332} C_VEL
LIN {X 0,Y 248.988,Z 1120.372,A -85,B 0,C 180,E1 20547.137,E2 20547.137} C_VEL
LIN {X 0,Y 246.326,Z 1134.789,A -85,B 0,C 180,E1 20554.432,E2 20554.432} C_VEL
LIN {X 0,Y 245.064,Z 1139.906,A -85,B 0,C 180,E1 20556.825,E2 20556.825} C_VEL
LIN {X 0,Y 230.734,Z 1157.967,A -85,B 0,C 180,E1 20561.925,E2 20561.925} C_VEL
LIN {X 0,Y 220.163,Z 1167.687,A -85,B 0,C 180,E1 20564.49,E2 20564.49} C_VEL
LIN {X 0,Y 209.681,Z 1176.533,A -85,B 0,C 180,E1 20567.395,E2 20567.395} C_VEL
LIN {X 0,Y 194.351,Z 1191.753,A -85,B 0,C 180,E1 20577.079,E2 20577.079} C_VEL
LIN {X 0,Y 183.696,Z 1201.973,A -85,B 0,C 180,E1 20588.307,E2 20588.307} C_VEL
LIN {X 0,Y 178.335,Z 1207.374,A -85,B 0,C 180,E1 20600.258,E2 20600.258} C_VEL
LIN {X 0,Y 177.666,Z 1208.61,A -85,B 0,C 180,E1 20610.002,E2 20610.002} C_VEL
LIN {X 0,Y 178.322,Z 1207.331,A -85,B 0,C 180,E1 20619.746,E2 20619.746} C_VEL
LIN {X 0,Y 183.739,Z 1201.869,A -85,B 0,C 180,E1 20631.691,E2 20631.691} C_VEL
LIN {X 0,Y 194.455,Z 1191.583,A -85,B 0,C 180,E1 20642.905,E2 20642.905} C_VEL
LIN {X 0,Y 210.477,Z 1175.605,A -85,B 0,C 180,E1 20652.932,E2 20652.932} C_VEL
LIN {X 0,Y 230.117,Z 1153.903,A -85,B 0,C 180,E1 20661.145,E2 20661.145} C_VEL
LIN {X 0,Y 238.273,Z 1143.916,A -85,B 0,C 180,E1 20663.852,E2 20663.852} C_VEL
LIN {X 0,Y 242.228,Z 1131.074,A -85,B 0,C 180,E1 20670.109,E2 20670.109} C_VEL
LIN {X 0,Y 244.651,Z 1118.169,A -85,B 0,C 180,E1 20677.702,E2 20677.702} C_VEL
LIN {X 0,Y 245.986,Z 1109.952,A -85,B 0,C 180,E1 20683.928,E2 20683.928} C_VEL
LIN {X 0,Y 247.079,Z 1105.027,A -85,B 0,C 180,E1 20689.443,E2 20689.443} C_VEL
LIN {X 0,Y 248.941,Z 1102.154,A -85,B 0,C 180,E1 20696.525,E2 20696.525} C_VEL
LIN {X 0,Y 250.198,Z 1102.068,A -85,B 0,C 180,E1 20700,E2 20700} C_VEL
LIN {X 0,Y 252.516,Z 1106.588,A -85,B 0,C 180,E1 20706.864,E2 20706.864} C_VEL
LIN {X 0,Y 255.984,Z 1117.157,A -85,B 0,C 180,E1 20714.509,E2 20714.509} C_VEL
LIN {X 0,Y 259.244,Z 1131.88,A -85,B 0,C 180,E1 20721.353,E2 20721.353} C_VEL
LIN {X 0,Y 260.469,Z 1141.086,A -85,B 0,C 180,E1 20724.754,E2 20724.754} C_VEL
LIN {X 0,Y 240.056,Z 1173.659,A -85,B 0,C 180,E1 20729.224,E2 20729.224} C_VEL
LIN {X 0,Y 219.453,Z 1202.086,A -85,B 0,C 180,E1 20735.379,E2 20735.379} C_VEL
LIN {X 0,Y 199.737,Z 1227.405,A -85,B 0,C 180,E1 20744.131,E2 20744.131} C_VEL
LIN {X 0,Y 184.998,Z 1247.241,A -85,B 0,C 180,E1 20755.179,E2 20755.179} C_VEL
LIN {X 0,Y 177.411,Z 1260.955,A -85,B 0,C 180,E1 20767.496,E2 20767.496} C_VEL
LIN {X 0,Y 176.14,Z 1268.984,A -85,B 0,C 180,E1 20780.132,E2 20780.132} C_VEL
LIN {X 0,Y 177.277,Z 1271.248,A -85,B 0,C 180,E1 20789.998,E2 20789.998} C_VEL
LIN {X 0,Y 176.097,Z 1268.993,A -85,B 0,C 180,E1 20799.867,E2 20799.867} C_VEL
LIN {X 0,Y 177.33,Z 1261.218,A -85,B 0,C 180,E1 20812.25,E2 20812.25} C_VEL
LIN {X 0,Y 184.966,Z 1247.292,A -85,B 0,C 180,E1 20824.824,E2 20824.824} C_VEL
LIN {X 0,Y 199.7,Z 1227.479,A -85,B 0,C 180,E1 20835.876,E2 20835.876} C_VEL
LIN {X 0,Y 219.371,Z 1202.245,A -85,B 0,C 180,E1 20844.619,E2 20844.619} C_VEL
LIN {X 0,Y 240.117,Z 1173.777,A -85,B 0,C 180,E1 20850.771,E2 20850.771} C_VEL
LIN {X 0,Y 260.153,Z 1142,A -85,B 0,C 180,E1 20855.143,E2 20855.143} C_VEL
LIN {X 0,Y 258.645,Z 1128.539,A -85,B 0,C 180,E1 20860.066,E2 20860.066} C_VEL
LIN {X 0,Y 255.646,Z 1115.898,A -85,B 0,C 180,E1 20866.343,E2 20866.343} C_VEL
LIN {X 0,Y 252.545,Z 1106.895,A -85,B 0,C 180,E1 20873.137,E2 20873.137} C_VEL
LIN {X 0,Y 250.214,Z 1102.433,A -85,B 0,C 180,E1 20880,E2 20880} C_VEL
LIN {X 0,Y 247.941,Z 1103.381,A -85,B 0,C 180,E1 20886.991,E2 20886.991} C_VEL
LIN {X 0,Y 246.471,Z 1108.239,A -85,B 0,C 180,E1 20894.175,E2 20894.175} C_VEL
LIN {X 0,Y 244.872,Z 1117.536,A -85,B 0,C 180,E1 20901.699,E2 20901.699} C_VEL
LIN {X 0,Y 242.419,Z 1130.457,A -85,B 0,C 180,E1 20909.372,E2 20909.372} C_VEL
LIN {X 0,Y 239.133,Z 1142.816,A -85,B 0,C 180,E1 20915.665,E2 20915.665} C_VEL
LIN {X 0,Y 219.264,Z 1166.366,A -85,B 0,C 180,E1 20922.947,E2 20922.947} C_VEL
LIN {X 0,Y 209.681,Z 1176.533,A -85,B 0,C 180,E1 20927.395,E2 20927.395} C_VEL
LIN {X 0,Y 199.422,Z 1184.465,A -85,B 0,C 180,E1 20930.711,E2 20930.711} C_VEL
LIN {X 0,Y 189.553,Z 1191.466,A -85,B 0,C 180,E1 20934.447,E2 20934.447} C_VEL
LIN {X 0,Y 178.202,Z 1201.684,A -85,B 0,C 180,E1 20944.953,E2 20944.953} C_VEL
LIN {X 0,Y 172.371,Z 1207.094,A -85,B 0,C 180,E1 20954.775,E2 20954.775} C_VEL
LIN {X 0,Y 169.892,Z 1209.703,A -85,B 0,C 180,E1 20964.906,E2 20964.906} C_VEL
LIN {X 0,Y 169.903,Z 1209.674,A -85,B 0,C 180,E1 20975.097,E2 20975.097} C_VEL
LIN {X 0,Y 173.366,Z 1206.116,A -85,B 0,C 180,E1 20987.477,E2 20987.477} C_VEL
LIN {X 0,Y 183.367,Z 1197.069,A -85,B 0,C 180,E1 21000.402,E2 21000.402} C_VEL
LIN {X 0,Y 199.331,Z 1182.261,A -85,B 0,C 180,E1 21011.63,E2 21011.63} C_VEL
LIN {X 0,Y 218.438,Z 1162.924,A -85,B 0,C 180,E1 21020.225,E2 21020.225} C_VEL
LIN {X 0,Y 233.1,Z 1145.782,A -85,B 0,C 180,E1 21025.422,E2 21025.422} C_VEL
LIN {X 0,Y 236.916,Z 1133.967,A -85,B 0,C 180,E1 21031.713,E2 21031.713} C_VEL
LIN {X 0,Y 239.908,Z 1121.442,A -85,B 0,C 180,E1 21039.763,E2 21039.763} C_VEL
LIN {X 0,Y 241.666,Z 1113.768,A -85,B 0,C 180,E1 21046.671,E2 21046.671} C_VEL
LIN {X 0,Y 243.395,Z 1109.723,A -85,B 0,C 180,E1 21053.223,E2 21053.223} C_VEL
LIN {X 0,Y 245.862,Z 1108.683,A -85,B 0,C 180,E1 21060,E2 21060} C_VEL
LIN {X 0,Y 248.129,Z 1113.401,A -85,B 0,C 180,E1 21066.986,E2 21066.986} C_VEL
LIN {X 0,Y 250.95,Z 1122.717,A -85,B 0,C 180,E1 21073.917,E2 21073.917} C_VEL
LIN {X 0,Y 253.537,Z 1135.748,A -85,B 0,C 180,E1 21080.326,E2 21080.326} C_VEL
LIN {X 0,Y 254.135,Z 1144.843,A -85,B 0,C 180,E1 21083.666,E2 21083.666} C_VEL
LIN {X 0,Y 231.865,Z 1178.165,A -85,B 0,C 180,E1 21088.523,E2 21088.523} C_VEL
LIN {X 0,Y 209.94,Z 1206.613,A -85,B 0,C 180,E1 21095.286,E2 21095.286} C_VEL
LIN {X 0,Y 190.316,Z 1230.386,A -85,B 0,C 180,E1 21104.468,E2 21104.468} C_VEL
LIN {X 0,Y 175.969,Z 1248.928,A -85,B 0,C 180,E1 21116.122,E2 21116.122} C_VEL
LIN {X 0,Y 169.07,Z 1261.528,A -85,B 0,C 180,E1 21129.081,E2 21129.081} C_VEL
LIN {X 0,Y 168.312,Z 1267.911,A -85,B 0,C 180,E1 21140.46,E2 21140.46} C_VEL
LIN {X 0,Y 169.483,Z 1269.872,A -85,B 0,C 180,E1 21149.998,E2 21149.998} C_VEL
LIN {X 0,Y 168.246,Z 1267.586,A -85,B 0,C 180,E1 21160.332,E2 21160.332} C_VEL
LIN {X 0,Y 169.432,Z 1260.584,A -85,B 0,C 180,E1 21172.24,E2 21172.24} C_VEL
LIN {X 0,Y 178.192,Z 1245.823,A -85,B 0,C 180,E1 21186.353,E2 21186.353} C_VEL
LIN {X 0,Y 193.994,Z 1226.011,A -85,B 0,C 180,E1 21197.642,E2 21197.642} C_VEL
LIN {X 0,Y 214.672,Z 1200.793,A -85,B 0,C 180,E1 21206.421,E2 21206.421} C_VEL
LIN {X 0,Y 236.785,Z 1171.509,A -85,B 0,C 180,E1 21212.648,E2 21212.648} C_VEL
LIN {X 0,Y 254.585,Z 1144.094,A -85,B 0,C 180,E1 21216.491,E2 21216.491} C_VEL
LIN {X 0,Y 252.293,Z 1128.417,A -85,B 0,C 180,E1 21223.131,E2 21223.131} C_VEL
LIN {X 0,Y 249.506,Z 1117.731,A -85,B 0,C 180,E1 21229.547,E2 21229.547} C_VEL
LIN {X 0,Y 246.899,Z 1110.846,A -85,B 0,C 180,E1 21236.496,E2 21236.496} C_VEL
LIN {X 0,Y 245.855,Z 1109.048,A -85,B 0,C 180,E1 21240,E2 21240} C_VEL
LIN {X 0,Y 243.388,Z 1110.124,A -85,B 0,C 180,E1 21247.26,E2 21247.26} C_VEL
LIN {X 0,Y 241.568,Z 1115,A -85,B 0,C 180,E1 21254.469,E2 21254.469} C_VEL
LIN {X 0,Y 239.641,Z 1123.088,A -85,B 0,C 180,E1 21261.226,E2 21261.226} C_VEL
LIN {X 0,Y 236.596,Z 1135.453,A -85,B 0,C 180,E1 21268.908,E2 21268.908} C_VEL
LIN {X 0,Y 233.136,Z 1146.143,A -85,B 0,C 180,E1 21274.656,E2 21274.656} C_VEL
LIN {X 0,Y 213.968,Z 1167.792,A -85,B 0,C 180,E1 21281.434,E2 21281.434} C_VEL
LIN {X 0,Y 195.497,Z 1185.983,A -85,B 0,C 180,E1 21290.52,E2 21290.52} C_VEL
LIN {X 0,Y 189.553,Z 1191.466,A -85,B 0,C 180,E1 21294.447,E2 21294.447} C_VEL
LIN {X 0,Y 180.172,Z 1197.607,A -85,B 0,C 180,E1 21298.637,E2 21298.637} C_VEL
LIN {X 0,Y 171.544,Z 1202.696,A -85,B 0,C 180,E1 21303.328,E2 21303.328} C_VEL
LIN {X 0,Y 164.847,Z 1208.472,A -85,B 0,C 180,E1 21314.062,E2 21314.062} C_VEL
LIN {X 0,Y 162.147,Z 1211.075,A -85,B 0,C 180,E1 21324.662,E2 21324.662} C_VEL
LIN {X 0,Y 162.156,Z 1211.047,A -85,B 0,C 180,E1 21335.342,E2 21335.342} C_VEL
LIN {X 0,Y 166.063,Z 1207.392,A -85,B 0,C 180,E1 21348.547,E2 21348.547} C_VEL
LIN {X 0,Y 177.168,Z 1197.975,A -85,B 0,C 180,E1 21362.166,E2 21362.166} C_VEL
LIN {X 0,Y 193.353,Z 1183.824,A -85,B 0,C 180,E1 21373.072,E2 21373.072} C_VEL
LIN {X 0,Y 213.396,Z 1164.439,A -85,B 0,C 180,E1 21381.791,E2 21381.791} C_VEL
LIN {X 0,Y 227.203,Z 1149.046,A -85,B 0,C 180,E1 21386.528,E2 21386.528} C_VEL
LIN {X 0,Y 231.734,Z 1136.832,A -85,B 0,C 180,E1 21393.465,E2 21393.465} C_VEL
LIN {X 0,Y 234.976,Z 1125.695,A -85,B 0,C 180,E1 21401.272,E2 21401.272} C_VEL
LIN {X 0,Y 237.481,Z 1118.322,A -85,B 0,C 180,E1 21409.011,E2 21409.011} C_VEL
LIN {X 0,Y 239.888,Z 1115.273,A -85,B 0,C 180,E1 21416.394,E2 21416.394} C_VEL
LIN {X 0,Y 241.45,Z 1115.38,A -85,B 0,C 180,E1 21420.281,E2 21420.281} C_VEL
LIN {X 0,Y 243.598,Z 1120.11,A -85,B 0,C 180,E1 21427.117,E2 21427.117} C_VEL
LIN {X 0,Y 246.155,Z 1129.655,A -85,B 0,C 180,E1 21434.194,E2 21434.194} C_VEL
LIN {X 0,Y 248.255,Z 1143.548,A -85,B 0,C 180,E1 21440.922,E2 21440.922} C_VEL
LIN {X 0,Y 248.216,Z 1147.702,A -85,B 0,C 180,E1 21442.468,E2 21442.468} C_VEL
LIN {X 0,Y 226.63,Z 1178.559,A -85,B 0,C 180,E1 21447.052,E2 21447.052} C_VEL
LIN {X 0,Y 204.097,Z 1206.506,A -85,B 0,C 180,E1 21453.812,E2 21453.812} C_VEL
LIN {X 0,Y 183.675,Z 1229.967,A -85,B 0,C 180,E1 21463.155,E2 21463.155} C_VEL
LIN {X 0,Y 168.874,Z 1247.812,A -85,B 0,C 180,E1 21474.844,E2 21474.844} C_VEL
LIN {X 0,Y 161.463,Z 1260.085,A -85,B 0,C 180,E1 21488.046,E2 21488.046} C_VEL
LIN {X 0,Y 160.405,Z 1266.16,A -85,B 0,C 180,E1 21499.153,E2 21499.153} C_VEL
LIN {X 0,Y 161.671,Z 1268.494,A -85,B 0,C 180,E1 21509.998,E2 21509.998} C_VEL
LIN {X 0,Y 160.384,Z 1266.175,A -85,B 0,C 180,E1 21520.844,E2 21520.844} C_VEL
LIN {X 0,Y 161.889,Z 1259.141,A -85,B 0,C 180,E1 21533.336,E2 21533.336} C_VEL
LIN {X 0,Y 171.549,Z 1244.353,A -85,B 0,C 180,E1 21548.004,E2 21548.004} C_VEL
LIN {X 0,Y 189.522,Z 1223.395,A -85,B 0,C 180,E1 21560,E2 21560} C_VEL
LIN {X 0,Y 210.374,Z 1199.157,A -85,B 0,C 180,E1 21568.342,E2 21568.342} C_VEL
LIN {X 0,Y 233.114,Z 1170.058,A -85,B 0,C 180,E1 21574.447,E2 21574.447} C_VEL
LIN {X 0,Y 248.314,Z 1147.839,A -85,B 0,C 180,E1 21577.521,E2 21577.521} C_VEL
LIN {X 0,Y 247.172,Z 1134.92,A -85,B 0,C 180,E1 21583.051,E2 21583.051} C_VEL
LIN {X 0,Y 244.912,Z 1124.52,A -85,B 0,C 180,E1 21589.348,E2 21589.348} C_VEL
LIN {X 0,Y 242.43,Z 1117.427,A -85,B 0,C 180,E1 21596.431,E2 21596.431} C_VEL
LIN {X 0,Y 241.41,Z 1115.573,A -85,B 0,C 180,E1 21600,E2 21600} C_VEL
LIN {X 0,Y 238.639,Z 1116.547,A -85,B 0,C 180,E1 21607.265,E2 21607.265} C_VEL
LIN {X 0,Y 236.956,Z 1119.945,A -85,B 0,C 180,E1 21612.878,E2 21612.878} C_VEL
LIN {X 0,Y 234.55,Z 1127.565,A -85,B 0,C 180,E1 21620.021,E2 21620.021} C_VEL
LIN {X 0,Y 230.912,Z 1139.524,A -85,B 0,C 180,E1 21627.964,E2 21627.964} C_VEL
LIN {X 0,Y 227.292,Z 1149.262,A -85,B 0,C 180,E1 21633.48,E2 21633.48} C_VEL
LIN {X 0,Y 206.134,Z 1171.882,A -85,B 0,C 180,E1 21640.895,E2 21640.895} C_VEL
LIN {X 0,Y 186.113,Z 1190.404,A -85,B 0,C 180,E1 21651.072,E2 21651.072} C_VEL
LIN {X 0,Y 171.544,Z 1202.696,A -85,B 0,C 180,E1 21663.328,E2 21663.328} C_VEL
LIN {X 0,Y 163.895,Z 1206.965,A -85,B 0,C 180,E1 21668.512,E2 21668.512} C_VEL
LIN {X 0,Y 156.946,Z 1210.159,A -85,B 0,C 180,E1 21674.183,E2 21674.183} C_VEL
LIN {X 0,Y 154.361,Z 1212.723,A -85,B 0,C 180,E1 21690.002,E2 21690.002} C_VEL
LIN {X 0,Y 155.299,Z 1211.463,A -85,B 0,C 180,E1 21701.208,E2 21701.208} C_VEL
LIN {X 0,Y 162.15,Z 1206.016,A -85,B 0,C 180,E1 21714.76,E2 21714.76} C_VEL
LIN {X 0,Y 175.14,Z 1195.745,A -85,B 0,C 180,E1 21727.096,E2 21727.096} C_VEL
LIN {X 0,Y 193.907,Z 1179.764,A -85,B 0,C 180,E1 21737.674,E2 21737.674} C_VEL
LIN {X 0,Y 215.019,Z 1159.286,A -85,B 0,C 180,E1 21745.635,E2 21745.635} C_VEL
LIN {X 0,Y 221.012,Z 1152.883,A -85,B 0,C 180,E1 21747.468,E2 21747.468} C_VEL
LIN {X 0,Y 225.448,Z 1142.857,A -85,B 0,C 180,E1 21753.264,E2 21753.264} C_VEL
LIN {X 0,Y 229.278,Z 1132.384,A -85,B 0,C 180,E1 21760.788,E2 21760.788} C_VEL
LIN {X 0,Y 231.872,Z 1125.699,A -85,B 0,C 180,E1 21767.479,E2 21767.479} C_VEL
LIN {X 0,Y 233.876,Z 1122.53,A -85,B 0,C 180,E1 21773.384,E2 21773.384} C_VEL
LIN {X 0,Y 236.691,Z 1121.578,A -85,B 0,C 180,E1 21780,E2 21780} C_VEL
LIN {X 0,Y 238.842,Z 1126.602,A -85,B 0,C 180,E1 21787.259,E2 21787.259} C_VEL
LIN {X 0,Y 241.148,Z 1136.558,A -85,B 0,C 180,E1 21794.495,E2 21794.495} C_VEL
LIN {X 0,Y 242.585,Z 1150.026,A -85,B 0,C 180,E1 21801.076,E2 21801.076} C_VEL
LIN {X 0,Y 218.663,Z 1182.639,A -85,B 0,C 180,E1 21806.212,E2 21806.212} C_VEL
LIN {X 0,Y 194.687,Z 1210.472,A -85,B 0,C 180,E1 21813.565,E2 21813.565} C_VEL
LIN {X 0,Y 174.103,Z 1232.747,A -85,B 0,C 180,E1 21823.511,E2 21823.511} C_VEL
LIN {X 0,Y 159.167,Z 1250.163,A -85,B 0,C 180,E1 21836.7,E2 21836.7} C_VEL
LIN {X 0,Y 152.994,Z 1261.101,A -85,B 0,C 180,E1 21850.816,E2 21850.816} C_VEL
LIN {X 0,Y 152.578,Z 1265.663,A -85,B 0,C 180,E1 21861.481,E2 21861.481} C_VEL
LIN {X 0,Y 153.869,Z 1267.117,A -85,B 0,C 180,E1 21869.998,E2 21869.998} C_VEL
LIN {X 0,Y 152.538,Z 1264.764,A -85,B 0,C 180,E1 21881.409,E2 21881.409} C_VEL
LIN {X 0,Y 154.392,Z 1257.694,A -85,B 0,C 180,E1 21894.542,E2 21894.542} C_VEL
LIN {X 0,Y 165.103,Z 1242.893,A -85,B 0,C 180,E1 21909.774,E2 21909.774} C_VEL
LIN {X 0,Y 183.947,Z 1222.282,A -85,B 0,C 180,E1 21921.832,E2 21921.832} C_VEL
LIN {X 0,Y 206.263,Z 1197.574,A -85,B 0,C 180,E1 21930.331,E2 21930.331} C_VEL
LIN {X 0,Y 229.681,Z 1168.607,A -85,B 0,C 180,E1 21936.302,E2 21936.302} C_VEL
LIN {X 0,Y 242.657,Z 1150.295,A -85,B 0,C 180,E1 21938.873,E2 21938.873} C_VEL
LIN {X 0,Y 241.207,Z 1136.74,A -85,B 0,C 180,E1 21945.509,E2 21945.509} C_VEL
LIN {X 0,Y 238.838,Z 1126.9,A -85,B 0,C 180,E1 21952.741,E2 21952.741} C_VEL
LIN {X 0,Y 236.668,Z 1121.931,A -85,B 0,C 180,E1 21960,E2 21960} C_VEL
LIN {X 0,Y 233.734,Z 1122.978,A -85,B 0,C 180,E1 21967.418,E2 21967.418} C_VEL
LIN {X 0,Y 231.489,Z 1127.076,A -85,B 0,C 180,E1 21973.871,E2 21973.871} C_VEL
LIN {X 0,Y 228.687,Z 1134.365,A -85,B 0,C 180,E1 21980.582,E2 21980.582} C_VEL
LIN {X 0,Y 224.579,Z 1145.327,A -85,B 0,C 180,E1 21988.056,E2 21988.056} C_VEL
LIN {X 0,Y 220.941,Z 1153.154,A -85,B 0,C 180,E1 21992.486,E2 21992.486} C_VEL
LIN {X 0,Y 198.144,Z 1176.012,A -85,B 0,C 180,E1 22000.399,E2 22000.399} C_VEL
LIN {X 0,Y 178.324,Z 1193.162,A -85,B 0,C 180,E1 22010.607,E2 22010.607} C_VEL
LIN {X 0,Y 164.115,Z 1204.452,A -85,B 0,C 180,E1 22022.632,E2 22022.632} C_VEL
LIN {X 0,Y 156.946,Z 1210.159,A -85,B 0,C 180,E1 22034.183,E2 22034.183} C_VEL
LIN {X 0,Y 151.046,Z 1212.578,A -85,B 0,C 180,E1 22040.239,E2 22040.239} C_VEL
LIN {X 0,Y 146.434,Z 1213.943,A -85,B 0,C 180,E1 22046.732,E2 22046.732} C_VEL
LIN {X 0,Y 146.668,Z 1213.794,A -85,B 0,C 180,E1 22055.907,E2 22055.907} C_VEL
LIN {X 0,Y 151.32,Z 1210.153,A -85,B 0,C 180,E1 22070.43,E2 22070.43} C_VEL
LIN {X 0,Y 164.081,Z 1200.75,A -85,B 0,C 180,E1 22085.088,E2 22085.088} C_VEL
LIN {X 0,Y 182.2,Z 1186.597,A -85,B 0,C 180,E1 22096.445,E2 22096.445} C_VEL
LIN {X 0,Y 204.881,Z 1166.428,A -85,B 0,C 180,E1 22105.511,E2 22105.511} C_VEL
LIN {X 0,Y 215.49,Z 1155.708,A -85,B 0,C 180,E1 22108.838,E2 22108.838} C_VEL
LIN {X 0,Y 220.752,Z 1144.794,A -85,B 0,C 180,E1 22115.787,E2 22115.787} C_VEL
LIN {X 0,Y 224.476,Z 1136.315,A -85,B 0,C 180,E1 22122.564,E2 22122.564} C_VEL
LIN {X 0,Y 227.039,Z 1131.093,A -85,B 0,C 180,E1 22128.499,E2 22128.499} C_VEL
LIN {X 0,Y 230.127,Z 1127.938,A -85,B 0,C 180,E1 22136.241,E2 22136.241} C_VEL
LIN {X 0,Y 231.875,Z 1127.878,A -85,B 0,C 180,E1 22140,E2 22140} C_VEL
LIN {X 0,Y 233.957,Z 1133.063,A -85,B 0,C 180,E1 22147.412,E2 22147.412} C_VEL
LIN {X 0,Y 235.861,Z 1143.263,A -85,B 0,C 180,E1 22154.827,E2 22154.827} C_VEL
LIN {X 0,Y 236.623,Z 1152.571,A -85,B 0,C 180,E1 22159.56,E2 22159.56} C_VEL
LIN {X 0,Y 232.643,Z 1158.915,A -85,B 0,C 180,E1 22160.646,E2 22160.646} C_VEL
LIN {X 0,Y 208.217,Z 1189.293,A -85,B 0,C 180,E1 22165.973,E2 22165.973} C_VEL
LIN {X 0,Y 182.792,Z 1216.734,A -85,B 0,C 180,E1 22174.354,E2 22174.354} C_VEL
LIN {X 0,Y 162.111,Z 1237.859,A -85,B 0,C 180,E1 22185.72,E2 22185.72} C_VEL
LIN {X 0,Y 149.144,Z 1252.812,A -85,B 0,C 180,E1 22199.607,E2 22199.607} C_VEL
LIN {X 0,Y 144.697,Z 1262.152,A -85,B 0,C 180,E1 22214.885,E2 22214.885} C_VEL
LIN {X 0,Y 145.055,Z 1265.005,A -85,B 0,C 180,E1 22224.027,E2 22224.027} C_VEL
LIN {X 0,Y 146.058,Z 1265.738,A -85,B 0,C 180,E1 22229.998,E2 22229.998} C_VEL
LIN {X 0,Y 144.681,Z 1263.348,A -85,B 0,C 180,E1 22242.038,E2 22242.038} C_VEL
LIN {X 0,Y 147.615,Z 1255.196,A -85,B 0,C 180,E1 22257.386,E2 22257.386} C_VEL
LIN {X 0,Y 158.837,Z 1241.435,A -85,B 0,C 180,E1 22271.682,E2 22271.682} C_VEL
LIN {X 0,Y 178.371,Z 1221.372,A -85,B 0,C 180,E1 22283.689,E2 22283.689} C_VEL
LIN {X 0,Y 202.279,Z 1196.145,A -85,B 0,C 180,E1 22292.357,E2 22292.357} C_VEL
LIN {X 0,Y 226.497,Z 1167.157,A -85,B 0,C 180,E1 22298.209,E2 22298.209} C_VEL
LIN {X 0,Y 235.838,Z 1154.576,A -85,B 0,C 180,E1 22299.978,E2 22299.978} C_VEL
LIN {X 0,Y 236.588,Z 1150.701,A -85,B 0,C 180,E1 22301.404,E2 22301.404} C_VEL
LIN {X 0,Y 235.306,Z 1139.175,A -85,B 0,C 180,E1 22307.823,E2 22307.823} C_VEL
LIN {X 0,Y 233.451,Z 1131.575,A -85,B 0,C 180,E1 22314.436,E2 22314.436} C_VEL
LIN {X 0,Y 231.847,Z 1128.205,A -85,B 0,C 180,E1 22320,E2 22320} C_VEL
LIN {X 0,Y 228.6,Z 1129.279,A -85,B 0,C 180,E1 22327.586,E2 22327.586} C_VEL
LIN {X 0,Y 225.962,Z 1133.413,A -85,B 0,C 180,E1 22334.218,E2 22334.218} C_VEL
LIN {X 0,Y 222.551,Z 1141.061,A -85,B 0,C 180,E1 22341.225,E2 22341.225} C_VEL
LIN {X 0,Y 217.321,Z 1152.45,A -85,B 0,C 180,E1 22349.08,E2 22349.08} C_VEL
LIN {X 0,Y 214.625,Z 1156.777,A -85,B 0,C 180,E1 22351.351,E2 22351.351} C_VEL
LIN {X 0,Y 192.76,Z 1177.723,A -85,B 0,C 180,E1 22358.774,E2 22358.774} C_VEL
LIN {X 0,Y 172.017,Z 1194.783,A -85,B 0,C 180,E1 22369.146,E2 22369.146} C_VEL
LIN {X 0,Y 157.185,Z 1205.837,A -85,B 0,C 180,E1 22381.316,E2 22381.316} C_VEL
LIN {X 0,Y 149.292,Z 1211.577,A -85,B 0,C 180,E1 22393.627,E2 22393.627} C_VEL
LIN {X 0,Y 146.434,Z 1213.943,A -85,B 0,C 180,E1 22406.732,E2 22406.732} C_VEL
LIN {X 0,Y 143.899,Z 1214.521,A -85,B 0,C 180,E1 22411.801,E2 22411.801} C_VEL
LIN {X 0,Y 139.471,Z 1214.648,A -85,B 0,C 180,E1 22420.356,E2 22420.356} C_VEL
LIN {X 0,Y 139.516,Z 1214.506,A -85,B 0,C 180,E1 22420.583,E2 22420.583} C_VEL
LIN {X 0,Y 145.877,Z 1210.201,A -85,B 0,C 180,E1 22434.445,E2 22434.445} C_VEL
LIN {X 0,Y 159.387,Z 1200.942,A -85,B 0,C 180,E1 22447.983,E2 22447.983} C_VEL
LIN {X 0,Y 179.118,Z 1186.205,A -85,B 0,C 180,E1 22459.31,E2 22459.31} C_VEL
LIN {X 0,Y 200.616,Z 1167.75,A -85,B 0,C 180,E1 22467.377,E2 22467.377} C_VEL
LIN {X 0,Y 210.114,Z 1158.363,A -85,B 0,C 180,E1 22470.427,E2 22470.427} C_VEL
LIN {X 0,Y 215.449,Z 1148.55,A -85,B 0,C 180,E1 22477.208,E2 22477.208} C_VEL
LIN {X 0,Y 219.562,Z 1140.572,A -85,B 0,C 180,E1 22484.201,E2 22484.201} C_VEL
LIN {X 0,Y 222.312,Z 1136.194,A -85,B 0,C 180,E1 22490.23,E2 22490.23} C_VEL
LIN {X 0,Y 225.037,Z 1134.139,A -85,B 0,C 180,E1 22496.155,E2 22496.155} C_VEL
LIN {X 0,Y 226.856,Z 1133.985,A -85,B 0,C 180,E1 22500,E2 22500} C_VEL
LIN {X 0,Y 228.851,Z 1139.329,A -85,B 0,C 180,E1 22507.578,E2 22507.578} C_VEL
LIN {X 0,Y 230.291,Z 1148.442,A -85,B 0,C 180,E1 22514.317,E2 22514.317} C_VEL
LIN {X 0,Y 230.659,Z 1155.52,A -85,B 0,C 180,E1 22518.174,E2 22518.174} C_VEL
LIN {X 0,Y 228.528,Z 1159.318,A -85,B 0,C 180,E1 22518.976,E2 22518.976} C_VEL
LIN {X 0,Y 202.79,Z 1189.976,A -85,B 0,C 180,E1 22524.381,E2 22524.381} C_VEL
LIN {X 0,Y 177.031,Z 1216.421,A -85,B 0,C 180,E1 22532.634,E2 22532.634} C_VEL
LIN {X 0,Y 155.885,Z 1236.733,A -85,B 0,C 180,E1 22543.84,E2 22543.84} C_VEL
LIN {X 0,Y 141.839,Z 1251.662,A -85,B 0,C 180,E1 22558.329,E2 22558.329} C_VEL
LIN {X 0,Y 136.925,Z 1260.728,A -85,B 0,C 180,E1 22574.005,E2 22574.005} C_VEL
LIN {X 0,Y 137.189,Z 1263.609,A -85,B 0,C 180,E1 22583.683,E2 22583.683} C_VEL
LIN {X 0,Y 138.246,Z 1264.36,A -85,B 0,C 180,E1 22589.998,E2 22589.998} C_VEL
LIN {X 0,Y 136.859,Z 1261.935,A -85,B 0,C 180,E1 22602.737,E2 22602.737} C_VEL
LIN {X 0,Y 140.25,Z 1253.915,A -85,B 0,C 180,E1 22618.7,E2 22618.7} C_VEL
LIN {X 0,Y 154.263,Z 1238.404,A -85,B 0,C 180,E1 22634.953,E2 22634.953} C_VEL
LIN {X 0,Y 174.695,Z 1218.763,A -85,B 0,C 180,E1 22646.41,E2 22646.41} C_VEL
LIN {X 0,Y 198.587,Z 1194.692,A -85,B 0,C 180,E1 22654.465,E2 22654.465} C_VEL
LIN {X 0,Y 222.78,Z 1166.712,A -85,B 0,C 180,E1 22660.019,E2 22660.019} C_VEL
LIN {X 0,Y 230.699,Z 1156.04,A -85,B 0,C 180,E1 22661.655,E2 22661.655} C_VEL
LIN {X 0,Y 229.805,Z 1144.138,A -85,B 0,C 180,E1 22668.639,E2 22668.639} C_VEL
LIN {X 0,Y 227.851,Z 1136.333,A -85,B 0,C 180,E1 22676.203,E2 22676.203} C_VEL
LIN {X 0,Y 226.372,Z 1134.302,A -85,B 0,C 180,E1 22680.858,E2 22680.858} C_VEL
LIN {X 0,Y 223.283,Z 1135.436,A -85,B 0,C 180,E1 22687.768,E2 22687.768} C_VEL
LIN {X 0,Y 220.601,Z 1139.141,A -85,B 0,C 180,E1 22693.911,E2 22693.911} C_VEL
LIN {X 0,Y 216.252,Z 1147.214,A -85,B 0,C 180,E1 22701.553,E2 22701.553} C_VEL
LIN {X 0,Y 210.723,Z 1157.629,A -85,B 0,C 180,E1 22708.948,E2 22708.948} C_VEL
LIN {X 0,Y 207.608,Z 1161.193,A -85,B 0,C 180,E1 22710.396,E2 22710.396} C_VEL
LIN {X 0,Y 184.673,Z 1181.843,A -85,B 0,C 180,E1 22718.225,E2 22718.225} C_VEL
LIN {X 0,Y 162.785,Z 1198.679,A -85,B 0,C 180,E1 22729.544,E2 22729.544} C_VEL
LIN {X 0,Y 147.975,Z 1208.888,A -85,B 0,C 180,E1 22742.686,E2 22742.686} C_VEL
LIN {X 0,Y 140.03,Z 1214.259,A -85,B 0,C 180,E1 22757.556,E2 22757.556} C_VEL
LIN {X 0,Y 138.818,Z 1215.466,A -85,B 0,C 180,E1 22770.002,E2 22770.002} C_VEL
LIN {X 0,Y 139.516,Z 1214.506,A -85,B 0,C 180,E1 22780.583,E2 22780.583} C_VEL
LIN {X 0,Y 138.068,Z 1213.682,A -85,B 0,C 180,E1 22787.795,E2 22787.795} C_VEL
LIN {X 0,Y 138.267,Z 1211.899,A -85,B 0,C 180,E1 22795.071,E2 22795.071} C_VEL
LIN {X 0,Y 153.268,Z 1202.331,A -85,B 0,C 180,E1 22809.792,E2 22809.792} C_VEL
LIN {X 0,Y 174.098,Z 1187.593,A -85,B 0,C 180,E1 22821.271,E2 22821.271} C_VEL
LIN {X 0,Y 197.81,Z 1167.949,A -85,B 0,C 180,E1 22829.701,E2 22829.701} C_VEL
LIN {X 0,Y 204.174,Z 1162.001,A -85,B 0,C 180,E1 22831.528,E2 22831.528} C_VEL
LIN {X 0,Y 209.761,Z 1153.081,A -85,B 0,C 180,E1 22838.055,E2 22838.055} C_VEL
LIN {X 0,Y 214.643,Z 1145.064,A -85,B 0,C 180,E1 22845.782,E2 22845.782} C_VEL
LIN {X 0,Y 218.483,Z 1140.78,A -85,B 0,C 180,E1 22853.792,E2 22853.792} C_VEL
LIN {X 0,Y 221.691,Z 1139.976,A -85,B 0,C 180,E1 22860,E2 22860} C_VEL
LIN {X 0,Y 223.555,Z 1145.517,A -85,B 0,C 180,E1 22867.758,E2 22867.758} C_VEL
LIN {X 0,Y 224.612,Z 1154.785,A -85,B 0,C 180,E1 22874.592,E2 22874.592} C_VEL
LIN {X 0,Y 224.175,Z 1160.167,A -85,B 0,C 180,E1 22877.321,E2 22877.321} C_VEL
LIN {X 0,Y 198.104,Z 1189.985,A -85,B 0,C 180,E1 22882.57,E2 22882.57} C_VEL
LIN {X 0,Y 172.849,Z 1214.809,A -85,B 0,C 180,E1 22890.251,E2 22890.251} C_VEL
LIN {X 0,Y 150.025,Z 1235.461,A -85,B 0,C 180,E1 22901.701,E2 22901.701} C_VEL
LIN {X 0,Y 135.12,Z 1249.888,A -85,B 0,C 180,E1 22916.052,E2 22916.052} C_VEL
LIN {X 0,Y 129.174,Z 1259.301,A -85,B 0,C 180,E1 22933.017,E2 22933.017} C_VEL
LIN {X 0,Y 129.327,Z 1262.212,A -85,B 0,C 180,E1 22943.297,E2 22943.297} C_VEL
LIN {X 0,Y 130.399,Z 1262.975,A -85,B 0,C 180,E1 22949.998,E2 22949.998} C_VEL
LIN {X 0,Y 129.019,Z 1260.515,A -85,B 0,C 180,E1 22963.526,E2 22963.526} C_VEL
LIN {X 0,Y 132.941,Z 1252.591,A -85,B 0,C 180,E1 22980.217,E2 22980.217} C_VEL
LIN {X 0,Y 146.816,Z 1238.498,A -85,B 0,C 180,E1 22996.009,E2 22996.009} C_VEL
LIN {X 0,Y 169.608,Z 1217.894,A -85,B 0,C 180,E1 23008.481,E2 23008.481} C_VEL
LIN {X 0,Y 195.161,Z 1193.233,A -85,B 0,C 180,E1 23016.659,E2 23016.659} C_VEL
LIN {X 0,Y 221.235,Z 1163.892,A -85,B 0,C 180,E1 23022.218,E2 23022.218} C_VEL
LIN {X 0,Y 224.792,Z 1159.026,A -85,B 0,C 180,E1 23023.098,E2 23023.098} C_VEL
LIN {X 0,Y 224.115,Z 1148.906,A -85,B 0,C 180,E1 23029.502,E2 23029.502} C_VEL
LIN {X 0,Y 222.658,Z 1142.393,A -85,B 0,C 180,E1 23036.114,E2 23036.114} C_VEL
LIN {X 0,Y 221.634,Z 1140.305,A -85,B 0,C 180,E1 23040,E2 23040} C_VEL
LIN {X 0,Y 217.859,Z 1141.504,A -85,B 0,C 180,E1 23047.962,E2 23047.962} C_VEL
LIN {X 0,Y 214.682,Z 1145.328,A -85,B 0,C 180,E1 23054.303,E2 23054.303} C_VEL
LIN {X 0,Y 209.735,Z 1153.346,A -85,B 0,C 180,E1 23061.936,E2 23061.936} C_VEL
LIN {X 0,Y 204.843,Z 1161.283,A -85,B 0,C 180,E1 23067.874,E2 23067.874} C_VEL
LIN {X 0,Y 186.344,Z 1178.079,A -85,B 0,C 180,E1 23073.9,E2 23073.9} C_VEL
LIN {X 0,Y 162.804,Z 1195.987,A -85,B 0,C 180,E1 23084.146,E2 23084.146} C_VEL
LIN {X 0,Y 146.444,Z 1206.808,A -85,B 0,C 180,E1 23095.518,E2 23095.518} C_VEL
LIN {X 0,Y 135.08,Z 1213.983,A -85,B 0,C 180,E1 23110.422,E2 23110.422} C_VEL
LIN {X 0,Y 131.164,Z 1216.571,A -85,B 0,C 180,E1 23123.396,E2 23123.396} C_VEL
LIN {X 0,Y 131.17,Z 1216.545,A -85,B 0,C 180,E1 23136.608,E2 23136.608} C_VEL
LIN {X 0,Y 138.267,Z 1211.899,A -85,B 0,C 180,E1 23155.071,E2 23155.071} C_VEL
LIN {X 0,Y 140.05,Z 1209.389,A -85,B 0,C 180,E1 23162.178,E2 23162.178} C_VEL
LIN {X 0,Y 143.527,Z 1206.079,A -85,B 0,C 180,E1 23169.02,E2 23169.02} C_VEL
LIN {X 0,Y 164.454,Z 1192.475,A -85,B 0,C 180,E1 23181.259,E2 23181.259} C_VEL
LIN {X 0,Y 190.437,Z 1172.449,A -85,B 0,C 180,E1 23190.653,E2 23190.653} C_VEL
LIN {X 0,Y 198.882,Z 1164.94,A -85,B 0,C 180,E1 23193.088,E2 23193.088} C_VEL
LIN {X 0,Y 204.465,Z 1156.864,A -85,B 0,C 180,E1 23199.48,E2 23199.48} C_VEL
LIN {X 0,Y 208.492,Z 1151.131,A -85,B 0,C 180,E1 23205.327,E2 23205.327} C_VEL
LIN {X 0,Y 212.753,Z 1146.705,A -85,B 0,C 180,E1 23213.224,E2 23213.224} C_VEL
LIN {X 0,Y 216.368,Z 1145.886,A -85,B 0,C 180,E1 23220,E2 23220} C_VEL
LIN {X 0,Y 217.742,Z 1149.674,A -85,B 0,C 180,E1 23225.967,E2 23225.967} C_VEL
LIN {X 0,Y 218.727,Z 1157.965,A -85,B 0,C 180,E1 23233,E2 23233} C_VEL
LIN {X 0,Y 218.212,Z 1163.108,A -85,B 0,C 180,E1 23235.882,E2 23235.882} C_VEL
LIN {X 0,Y 191.994,Z 1191.601,A -85,B 0,C 180,E1 23241.034,E2 23241.034} C_VEL
LIN {X 0,Y 165.875,Z 1215.906,A -85,B 0,C 180,E1 23248.878,E2 23248.878} C_VEL
LIN {X 0,Y 142.34,Z 1235.914,A -85,B 0,C 180,E1 23260.725,E2 23260.725} C_VEL
LIN {X 0,Y 126.731,Z 1250.126,A -85,B 0,C 180,E1 23276.457,E2 23276.457} C_VEL
LIN {X 0,Y 121.453,Z 1257.872,A -85,B 0,C 180,E1 23291.901,E2 23291.901} C_VEL
LIN {X 0,Y 121.531,Z 1260.919,A -85,B 0,C 180,E1 23303.359,E2 23303.359} C_VEL
LIN {X 0,Y 122.577,Z 1261.595,A -85,B 0,C 180,E1 23309.997,E2 23309.997} C_VEL
LIN {X 0,Y 121.214,Z 1259.096,A -85,B 0,C 180,E1 23324.415,E2 23324.415} C_VEL
LIN {X 0,Y 125.417,Z 1251.625,A -85,B 0,C 180,E1 23341.277,E2 23341.277} C_VEL
LIN {X 0,Y 141.142,Z 1237.025,A -85,B 0,C 180,E1 23358.449,E2 23358.449} C_VEL
LIN {X 0,Y 164.547,Z 1217.212,A -85,B 0,C 180,E1 23370.597,E2 23370.597} C_VEL
LIN {X 0,Y 190.496,Z 1193.336,A -85,B 0,C 180,E1 23378.551,E2 23378.551} C_VEL
LIN {X 0,Y 217.198,Z 1164.482,A -85,B 0,C 180,E1 23383.977,E2 23383.977} C_VEL
LIN {X 0,Y 218.817,Z 1161.436,A -85,B 0,C 180,E1 23384.895,E2 23384.895} C_VEL
LIN {X 0,Y 218.331,Z 1152.884,A -85,B 0,C 180,E1 23391.054,E2 23391.054} C_VEL
LIN {X 0,Y 216.771,Z 1147.177,A -85,B 0,C 180,E1 23398.005,E2 23398.005} C_VEL
LIN {X 0,Y 216.317,Z 1146.207,A -85,B 0,C 180,E1 23400,E2 23400} C_VEL
LIN {X 0,Y 212.773,Z 1146.929,A -85,B 0,C 180,E1 23406.844,E2 23406.844} C_VEL
LIN {X 0,Y 208.569,Z 1151.311,A -85,B 0,C 180,E1 23414.668,E2 23414.668} C_VEL
LIN {X 0,Y 203.422,Z 1158.623,A -85,B 0,C 180,E1 23421.77,E2 23421.77} C_VEL
LIN {X 0,Y 198.475,Z 1165.52,A -85,B 0,C 180,E1 23426.966,E2 23426.966} C_VEL
LIN {X 0,Y 172.521,Z 1186.806,A -85,B 0,C 180,E1 23435.282,E2 23435.282} C_VEL
LIN {X 0,Y 149.162,Z 1202.665,A -85,B 0,C 180,E1 23446.935,E2 23446.935} C_VEL
LIN {X 0,Y 131.757,Z 1213.041,A -85,B 0,C 180,E1 23462.737,E2 23462.737} C_VEL
LIN {X 0,Y 124.85,Z 1217.01,A -85,B 0,C 180,E1 23476.014,E2 23476.014} C_VEL
LIN {X 0,Y 123.277,Z 1218.208,A -85,B 0,C 180,E1 23490.002,E2 23490.002} C_VEL
LIN {X 0,Y 125.426,Z 1216.605,A -85,B 0,C 180,E1 23505.753,E2 23505.753} C_VEL
LIN {X 0,Y 134.288,Z 1211.559,A -85,B 0,C 180,E1 23520.379,E2 23520.379} C_VEL
LIN {X 0,Y 143.527,Z 1206.079,A -85,B 0,C 180,E1 23529.02,E2 23529.02} C_VEL
LIN {X 0,Y 148.555,Z 1202.049,A -85,B 0,C 180,E1 23535.429,E2 23535.429} C_VEL
LIN {X 0,Y 154.865,Z 1196.945,A -85,B 0,C 180,E1 23541.314,E2 23541.314} C_VEL
LIN {X 0,Y 179.57,Z 1179.505,A -85,B 0,C 180,E1 23550.679,E2 23550.679} C_VEL
LIN {X 0,Y 193.933,Z 1167.55,A -85,B 0,C 180,E1 23555.058,E2 23555.058} C_VEL
LIN {X 0,Y 200.388,Z 1159.21,A -85,B 0,C 180,E1 23562.47,E2 23562.47} C_VEL
LIN {X 0,Y 204.925,Z 1154.048,A -85,B 0,C 180,E1 23569.392,E2 23569.392} C_VEL
LIN {X 0,Y 208.558,Z 1151.775,A -85,B 0,C 180,E1 23575.851,E2 23575.851} C_VEL
LIN {X 0,Y 210.821,Z 1151.596,A -85,B 0,C 180,E1 23580,E2 23580} C_VEL
LIN {X 0,Y 212.138,Z 1155.492,A -85,B 0,C 180,E1 23586.125,E2 23586.125} C_VEL
LIN {X 0,Y 212.792,Z 1162.541,A -85,B 0,C 180,E1 23592.283,E2 23592.283} C_VEL
LIN {X 0,Y 212.763,Z 1165.115,A -85,B 0,C 180,E1 23593.987,E2 23593.987} C_VEL
LIN {X 0,Y 207.325,Z 1171.591,A -85,B 0,C 180,E1 23595.208,E2 23595.208} C_VEL
LIN {X 0,Y 181.187,Z 1197.739,A -85,B 0,C 180,E1 23600.641,E2 23600.641} C_VEL
LIN {X 0,Y 153.986,Z 1220.976,A -85,B 0,C 180,E1 23609.338,E2 23609.338} C_VEL
LIN {X 0,Y 131.706,Z 1238.65,A -85,B 0,C 180,E1 23621.86,E2 23621.86} C_VEL
LIN {X 0,Y 117.219,Z 1251.386,A -85,B 0,C 180,E1 23639.004,E2 23639.004} C_VEL
LIN {X 0,Y 113.405,Z 1257.648,A -85,B 0,C 180,E1 23654.563,E2 23654.563} C_VEL
LIN {X 0,Y 114.723,Z 1260.209,A -85,B 0,C 180,E1 23669.997,E2 23669.997} C_VEL
LIN {X 0,Y 113.415,Z 1257.672,A -85,B 0,C 180,E1 23685.43,E2 23685.43} C_VEL
LIN {X 0,Y 118.433,Z 1250.167,A -85,B 0,C 180,E1 23703.352,E2 23703.352} C_VEL
LIN {X 0,Y 135.758,Z 1235.556,A -85,B 0,C 180,E1 23721.082,E2 23721.082} C_VEL
LIN {X 0,Y 162.04,Z 1214.557,A -85,B 0,C 180,E1 23733.676,E2 23733.676} C_VEL
LIN {X 0,Y 188.899,Z 1190.654,A -85,B 0,C 180,E1 23741.175,E2 23741.175} C_VEL
LIN {X 0,Y 212.27,Z 1166.314,A -85,B 0,C 180,E1 23745.635,E2 23745.635} C_VEL
LIN {X 0,Y 212.713,Z 1159.979,A -85,B 0,C 180,E1 23749.785,E2 23749.785} C_VEL
LIN {X 0,Y 211.674,Z 1153.735,A -85,B 0,C 180,E1 23756.4,E2 23756.4} C_VEL
LIN {X 0,Y 210.776,Z 1151.882,A -85,B 0,C 180,E1 23760,E2 23760} C_VEL
LIN {X 0,Y 208.618,Z 1151.966,A -85,B 0,C 180,E1 23764.148,E2 23764.148} C_VEL
LIN {X 0,Y 205.015,Z 1154.207,A -85,B 0,C 180,E1 23770.603,E2 23770.603} C_VEL
LIN {X 0,Y 200.384,Z 1159.45,A -85,B 0,C 180,E1 23777.53,E2 23777.53} C_VEL
LIN {X 0,Y 193.55,Z 1168.214,A -85,B 0,C 180,E1 23785.257,E2 23785.257} C_VEL
LIN {X 0,Y 166.345,Z 1189.383,A -85,B 0,C 180,E1 23793.759,E2 23793.759} C_VEL
LIN {X 0,Y 143.512,Z 1204.053,A -85,B 0,C 180,E1 23804.788,E2 23804.788} C_VEL
LIN {X 0,Y 127.505,Z 1213.043,A -85,B 0,C 180,E1 23817.823,E2 23817.823} C_VEL
LIN {X 0,Y 117.305,Z 1218.384,A -85,B 0,C 180,E1 23835.094,E2 23835.094} C_VEL
LIN {X 0,Y 115.49,Z 1219.582,A -85,B 0,C 180,E1 23850.003,E2 23850.003} C_VEL
LIN {X 0,Y 117.277,Z 1218.349,A -85,B 0,C 180,E1 23864.915,E2 23864.915} C_VEL
LIN {X 0,Y 127.572,Z 1212.946,A -85,B 0,C 180,E1 23882.163,E2 23882.163} C_VEL
LIN {X 0,Y 145.721,Z 1202.689,A -85,B 0,C 180,E1 23896.462,E2 23896.462} C_VEL
LIN {X 0,Y 154.865,Z 1196.945,A -85,B 0,C 180,E1 23901.314,E2 23901.314} C_VEL
LIN {X 0,Y 162.411,Z 1191.146,A -85,B 0,C 180,E1 23906.633,E2 23906.633} C_VEL
LIN {X 0,Y 169.521,Z 1185.534,A -85,B 0,C 180,E1 23910.931,E2 23910.931} C_VEL
LIN {X 0,Y 170.899,Z 1184.547,A -85,B 0,C 180,E1 23911.404,E2 23911.404} C_VEL
LIN {X 0,Y 188.265,Z 1171.064,A -85,B 0,C 180,E1 23916.375,E2 23916.375} C_VEL
LIN {X 0,Y 194.796,Z 1163.758,A -85,B 0,C 180,E1 23923.432,E2 23923.432} C_VEL
LIN {X 0,Y 199.306,Z 1159.345,A -85,B 0,C 180,E1 23929.833,E2 23929.833} C_VEL
LIN {X 0,Y 202.716,Z 1157.374,A -85,B 0,C 180,E1 23935.731,E2 23935.731} C_VEL
LIN {X 0,Y 205.187,Z 1157.233,A -85,B 0,C 180,E1 23940,E2 23940} C_VEL
LIN {X 0,Y 206.563,Z 1162.198,A -85,B 0,C 180,E1 23947.345,E2 23947.345} C_VEL
LIN {X 0,Y 206.668,Z 1168.512,A -85,B 0,C 180,E1 23952.653,E2 23952.653} C_VEL
LIN {X 0,Y 178.249,Z 1196.434,A -85,B 0,C 180,E1 23958.189,E2 23958.189} C_VEL
LIN {X 0,Y 149.477,Z 1219.946,A -85,B 0,C 180,E1 23966.773,E2 23966.773} C_VEL
LIN {X 0,Y 124.223,Z 1238.738,A -85,B 0,C 180,E1 23980.6,E2 23980.6} C_VEL
LIN {X 0,Y 108.372,Z 1251.891,A -85,B 0,C 180,E1 24000.83,E2 24000.83} C_VEL
LIN {X 0,Y 105.646,Z 1256.223,A -85,B 0,C 180,E1 24013.398,E2 24013.398} C_VEL
LIN {X 0,Y 106.886,Z 1258.826,A -85,B 0,C 180,E1 24029.997,E2 24029.997} C_VEL
LIN {X 0,Y 105.658,Z 1256.248,A -85,B 0,C 180,E1 24046.594,E2 24046.594} C_VEL
LIN {X 0,Y 111.731,Z 1248.612,A -85,B 0,C 180,E1 24065.874,E2 24065.874} C_VEL
LIN {X 0,Y 130.682,Z 1234.086,A -85,B 0,C 180,E1 24083.927,E2 24083.927} C_VEL
LIN {X 0,Y 158.511,Z 1213.083,A -85,B 0,C 180,E1 24096.385,E2 24096.385} C_VEL
LIN {X 0,Y 187.204,Z 1188.417,A -85,B 0,C 180,E1 24103.757,E2 24103.757} C_VEL
LIN {X 0,Y 206.735,Z 1168.636,A -85,B 0,C 180,E1 24107.351,E2 24107.351} C_VEL
LIN {X 0,Y 206.448,Z 1161.422,A -85,B 0,C 180,E1 24113.706,E2 24113.706} C_VEL
LIN {X 0,Y 205.149,Z 1157.485,A -85,B 0,C 180,E1 24120,E2 24120} C_VEL
LIN {X 0,Y 202.758,Z 1157.563,A -85,B 0,C 180,E1 24124.268,E2 24124.268} C_VEL
LIN {X 0,Y 199.328,Z 1159.551,A -85,B 0,C 180,E1 24130.218,E2 24130.218} C_VEL
LIN {X 0,Y 194.791,Z 1164.002,A -85,B 0,C 180,E1 24136.591,E2 24136.591} C_VEL
LIN {X 0,Y 188.194,Z 1171.32,A -85,B 0,C 180,E1 24143.634,E2 24143.634} C_VEL
LIN {X 0,Y 163.138,Z 1190.107,A -85,B 0,C 180,E1 24151.1,E2 24151.1} C_VEL
LIN {X 0,Y 138.086,Z 1205.439,A -85,B 0,C 180,E1 24162.472,E2 24162.472} C_VEL
LIN {X 0,Y 120.942,Z 1214.425,A -85,B 0,C 180,E1 24175.845,E2 24175.845} C_VEL
LIN {X 0,Y 109.697,Z 1219.813,A -85,B 0,C 180,E1 24194.342,E2 24194.342} C_VEL
LIN {X 0,Y 107.723,Z 1220.953,A -85,B 0,C 180,E1 24210.003,E2 24210.003} C_VEL
LIN {X 0,Y 109.761,Z 1219.725,A -85,B 0,C 180,E1 24225.963,E2 24225.963} C_VEL
LIN {X 0,Y 121.01,Z 1214.329,A -85,B 0,C 180,E1 24244.139,E2 24244.139} C_VEL
LIN {X 0,Y 142.287,Z 1202.958,A -85,B 0,C 180,E1 24259.823,E2 24259.823} C_VEL
LIN {X 0,Y 168.188,Z 1186.455,A -85,B 0,C 180,E1 24270.535,E2 24270.535} C_VEL
LIN {X 0,Y 170.899,Z 1184.547,A -85,B 0,C 180,E1 24271.404,E2 24271.404} C_VEL
LIN {X 0,Y 178.971,Z 1178.102,A -85,B 0,C 180,E1 24275.136,E2 24275.136} C_VEL
LIN {X 0,Y 185.754,Z 1171.511,A -85,B 0,C 180,E1 24280.751,E2 24280.751} C_VEL
LIN {X 0,Y 190.622,Z 1166.821,A -85,B 0,C 180,E1 24286.262,E2 24286.262} C_VEL
LIN {X 0,Y 193.939,Z 1164.128,A -85,B 0,C 180,E1 24291.048,E2 24291.048} C_VEL
LIN {X 0,Y 196.756,Z 1162.897,A -85,B 0,C 180,E1 24295.602,E2 24295.602} C_VEL
LIN {X 0,Y 199.324,Z 1162.661,A -85,B 0,C 180,E1 24300,E2 24300} C_VEL
LIN {X 0,Y 200.522,Z 1166.741,A -85,B 0,C 180,E1 24306.481,E2 24306.481} C_VEL
LIN {X 0,Y 200.681,Z 1171.45,A -85,B 0,C 180,E1 24310.887,E2 24310.887} C_VEL
LIN {X 0,Y 193.109,Z 1179.26,A -85,B 0,C 180,E1 24312.362,E2 24312.362} C_VEL
LIN {X 0,Y 163.227,Z 1205.415,A -85,B 0,C 180,E1 24318.588,E2 24318.588} C_VEL
LIN {X 0,Y 134.44,Z 1226.731,A -85,B 0,C 180,E1 24328.616,E2 24328.616} C_VEL
LIN {X 0,Y 111.594,Z 1242.347,A -85,B 0,C 180,E1 24343.745,E2 24343.745} C_VEL
LIN {X 0,Y 98.75,Z 1253.282,A -85,B 0,C 180,E1 24366.468,E2 24366.468} C_VEL
LIN {X 0,Y 97.771,Z 1256.592,A -85,B 0,C 180,E1 24381.118,E2 24381.118} C_VEL
LIN {X 0,Y 99.039,Z 1257.441,A -85,B 0,C 180,E1 24389.997,E2 24389.997} C_VEL
LIN {X 0,Y 97.929,Z 1254.82,A -85,B 0,C 180,E1 24407.947,E2 24407.947} C_VEL
LIN {X 0,Y 105.147,Z 1247.155,A -85,B 0,C 180,E1 24428.513,E2 24428.513} C_VEL
LIN {X 0,Y 125.938,Z 1232.611,A -85,B 0,C 180,E1 24447.004,E2 24447.004} C_VEL
LIN {X 0,Y 153.835,Z 1212.812,A -85,B 0,C 180,E1 24458.724,E2 24458.724} C_VEL
LIN {X 0,Y 183.379,Z 1188.519,A -85,B 0,C 180,E1 24465.892,E2 24465.892} C_VEL
LIN {X 0,Y 200.019,Z 1172.661,A -85,B 0,C 180,E1 24468.737,E2 24468.737} C_VEL
LIN {X 0,Y 200.712,Z 1169.022,A -85,B 0,C 180,E1 24471.352,E2 24471.352} C_VEL
LIN {X 0,Y 199.771,Z 1163.926,A -85,B 0,C 180,E1 24477.836,E2 24477.836} C_VEL
LIN {X 0,Y 199.292,Z 1162.909,A -85,B 0,C 180,E1 24480,E2 24480} C_VEL
LIN {X 0,Y 196.76,Z 1163.088,A -85,B 0,C 180,E1 24484.454,E2 24484.454} C_VEL
LIN {X 0,Y 192.876,Z 1165.098,A -85,B 0,C 180,E1 24490.564,E2 24490.564} C_VEL
LIN {X 0,Y 187.908,Z 1169.521,A -85,B 0,C 180,E1 24496.901,E2 24496.901} C_VEL
LIN {X 0,Y 182.582,Z 1174.773,A -85,B 0,C 180,E1 24502.075,E2 24502.075} C_VEL
LIN {X 0,Y 156.306,Z 1193.319,A -85,B 0,C 180,E1 24509.675,E2 24509.675} C_VEL
LIN {X 0,Y 130.593,Z 1208.009,A -85,B 0,C 180,E1 24521.32,E2 24521.32} C_VEL
LIN {X 0,Y 111.393,Z 1217.185,A -85,B 0,C 180,E1 24537.192,E2 24537.192} C_VEL
LIN {X 0,Y 102.308,Z 1221.136,A -85,B 0,C 180,E1 24552.846,E2 24552.846} C_VEL
LIN {X 0,Y 99.934,Z 1222.328,A -85,B 0,C 180,E1 24570.003,E2 24570.003} C_VEL
LIN {X 0,Y 102.277,Z 1221.104,A -85,B 0,C 180,E1 24587.166,E2 24587.166} C_VEL
LIN {X 0,Y 114.592,Z 1215.717,A -85,B 0,C 180,E1 24606.344,E2 24606.344} C_VEL
LIN {X 0,Y 135.381,Z 1205.464,A -85,B 0,C 180,E1 24621.287,E2 24621.287} C_VEL
LIN {X 0,Y 162.699,Z 1189.052,A -85,B 0,C 180,E1 24632.372,E2 24632.372} C_VEL
LIN {X 0,Y 182.715,Z 1174.501,A -85,B 0,C 180,E1 24637.859,E2 24637.859} C_VEL
LIN {X 0,Y 185.754,Z 1171.511,A -85,B 0,C 180,E1 24640.751,E2 24640.751} C_VEL
LIN {X 0,Y 187.418,Z 1169.647,A -85,B 0,C 180,E1 24644.694,E2 24644.694} C_VEL
LIN {X 0,Y 187.945,Z 1169.328,A -85,B 0,C 180,E1 24651.583,E2 24651.583} C_VEL
LIN {X 0,Y 193.36,Z 1167.956,A -85,B 0,C 180,E1 24660,E2 24660} C_VEL
LIN {X 0,Y 194.487,Z 1172.122,A -85,B 0,C 180,E1 24666.683,E2 24666.683} C_VEL
LIN {X 0,Y 194.491,Z 1174.708,A -85,B 0,C 180,E1 24669.292,E2 24669.292} C_VEL
LIN {X 0,Y 164.07,Z 1201.369,A -85,B 0,C 180,E1 24675.038,E2 24675.038} C_VEL
LIN {X 0,Y 134.432,Z 1222.702,A -85,B 0,C 180,E1 24683.858,E2 24683.858} C_VEL
LIN {X 0,Y 108.831,Z 1239.061,A -85,B 0,C 180,E1 24698.106,E2 24698.106} C_VEL
LIN {X 0,Y 92.436,Z 1250.618,A -85,B 0,C 180,E1 24720.672,E2 24720.672} C_VEL
LIN {X 0,Y 89.867,Z 1255.178,A -85,B 0,C 180,E1 24740.33,E2 24740.33} C_VEL
LIN {X 0,Y 91.155,Z 1256.05,A -85,B 0,C 180,E1 24749.997,E2 24749.997} C_VEL
LIN {X 0,Y 90.227,Z 1253.386,A -85,B 0,C 180,E1 24769.538,E2 24769.538} C_VEL
LIN {X 0,Y 99.817,Z 1244.985,A -85,B 0,C 180,E1 24792.857,E2 24792.857} C_VEL
LIN {X 0,Y 121.589,Z 1231.137,A -85,B 0,C 180,E1 24810.309,E2 24810.309} C_VEL
LIN {X 0,Y 152.119,Z 1210.51,A -85,B 0,C 180,E1 24821.989,E2 24821.989} C_VEL
LIN {X 0,Y 183.155,Z 1185.606,A -85,B 0,C 180,E1 24828.707,E2 24828.707} C_VEL
LIN {X 0,Y 194.519,Z 1174.872,A -85,B 0,C 180,E1 24830.701,E2 24830.701} C_VEL
LIN {X 0,Y 193.861,Z 1169.184,A -85,B 0,C 180,E1 24837.769,E2 24837.769} C_VEL
LIN {X 0,Y 193.309,Z 1168.197,A -85,B 0,C 180,E1 24840,E2 24840} C_VEL
LIN {X 0,Y 190.557,Z 1168.371,A -85,B 0,C 180,E1 24844.542,E2 24844.542} C_VEL
LIN {X 0,Y 185.273,Z 1171.247,A -85,B 0,C 180,E1 24852.219,E2 24852.219} C_VEL
LIN {X 0,Y 179.645,Z 1175.973,A -85,B 0,C 180,E1 24858.316,E2 24858.316} C_VEL
LIN {X 0,Y 177.062,Z 1178.252,A -85,B 0,C 180,E1 24860.373,E2 24860.373} C_VEL
LIN {X 0,Y 146.797,Z 1198.178,A -85,B 0,C 180,E1 24869.105,E2 24869.105} C_VEL
LIN {X 0,Y 120.801,Z 1211.681,A -85,B 0,C 180,E1 24881.456,E2 24881.456} C_VEL
LIN {X 0,Y 101.787,Z 1219.879,A -85,B 0,C 180,E1 24898.746,E2 24898.746} C_VEL
LIN {X 0,Y 92.57,Z 1223.445,A -85,B 0,C 180,E1 24920.622,E2 24920.622} C_VEL
LIN {X 0,Y 92.166,Z 1223.698,A -85,B 0,C 180,E1 24930.003,E2 24930.003} C_VEL
LIN {X 0,Y 94.859,Z 1222.479,A -85,B 0,C 180,E1 24948.555,E2 24948.555} C_VEL
LIN {X 0,Y 108.257,Z 1217.155,A -85,B 0,C 180,E1 24968.69,E2 24968.69} C_VEL
LIN {X 0,Y 130.604,Z 1206.854,A -85,B 0,C 180,E1 24983.982,E2 24983.982} C_VEL
LIN {X 0,Y 159.22,Z 1190.435,A -85,B 0,C 180,E1 24994.869,E2 24994.869} C_VEL
LIN {X 0,Y 177.173,Z 1177.999,A -85,B 0,C 180,E1 24999.54,E2 24999.54} C_VEL
LIN {X 0,Y 183.58,Z 1172.413,A -85,B 0,C 180,E1 25005.724,E2 25005.724} C_VEL
LIN {X 0,Y 187.945,Z 1169.328,A -85,B 0,C 180,E1 25011.583,E2 25011.583} C_VEL
LIN {X 0,Y 188.433,Z 1170.021,A -85,B 0,C 180,E1 25015.561,E2 25015.561} C_VEL
LIN {X 0,Y 187.845,Z 1174.048,A -85,B 0,C 180,E1 25022.258,E2 25022.258} C_VEL
LIN {X 0,Y 188.297,Z 1177.64,A -85,B 0,C 180,E1 25027.177,E2 25027.177} C_VEL
LIN {X 0,Y 186.916,Z 1179.465,A -85,B 0,C 180,E1 25027.987,E2 25027.987} C_VEL
LIN {X 0,Y 155.301,Z 1204.991,A -85,B 0,C 180,E1 25033.662,E2 25033.662} C_VEL
LIN {X 0,Y 123.48,Z 1226.081,A -85,B 0,C 180,E1 25043.567,E2 25043.567} C_VEL
LIN {X 0,Y 97.846,Z 1241.096,A -85,B 0,C 180,E1 25059.541,E2 25059.541} C_VEL
LIN {X 0,Y 83.288,Z 1251.091,A -85,B 0,C 180,E1 25084.939,E2 25084.939} C_VEL
LIN {X 0,Y 81.967,Z 1253.762,A -85,B 0,C 180,E1 25099.388,E2 25099.388} C_VEL
LIN {X 0,Y 83.276,Z 1254.659,A -85,B 0,C 180,E1 25109.996,E2 25109.996} C_VEL
LIN {X 0,Y 82.607,Z 1251.951,A -85,B 0,C 180,E1 25131.425,E2 25131.425} C_VEL
LIN {X 0,Y 93.897,Z 1243.517,A -85,B 0,C 180,E1 25156.314,E2 25156.314} C_VEL
LIN {X 0,Y 117.691,Z 1229.671,A -85,B 0,C 180,E1 25173.829,E2 25173.829} C_VEL
LIN {X 0,Y 149.717,Z 1209.081,A -85,B 0,C 180,E1 25184.996,E2 25184.996} C_VEL
LIN {X 0,Y 181.869,Z 1184.024,A -85,B 0,C 180,E1 25191.279,E2 25191.279} C_VEL
LIN {X 0,Y 186.619,Z 1179.894,A -85,B 0,C 180,E1 25191.963,E2 25191.963} C_VEL
LIN {X 0,Y 188.331,Z 1177.98,A -85,B 0,C 180,E1 25192.626,E2 25192.626} C_VEL
LIN {X 0,Y 187.807,Z 1174.306,A -85,B 0,C 180,E1 25197.698,E2 25197.698} C_VEL
LIN {X 0,Y 187.193,Z 1173.367,A -85,B 0,C 180,E1 25200,E2 25200} C_VEL
LIN {X 0,Y 182.487,Z 1174.165,A -85,B 0,C 180,E1 25207.13,E2 25207.13} C_VEL
LIN {X 0,Y 178.252,Z 1176.671,A -85,B 0,C 180,E1 25212.708,E2 25212.708} C_VEL
LIN {X 0,Y 172.648,Z 1180.964,A -85,B 0,C 180,E1 25218.248,E2 25218.248} C_VEL
LIN {X 0,Y 143.145,Z 1199.561,A -85,B 0,C 180,E1 25226.36,E2 25226.36} C_VEL
LIN {X 0,Y 115.752,Z 1213.066,A -85,B 0,C 180,E1 25238.542,E2 25238.542} C_VEL
LIN {X 0,Y 95.187,Z 1221.258,A -85,B 0,C 180,E1 25256.303,E2 25256.303} C_VEL
LIN {X 0,Y 84.89,Z 1224.821,A -85,B 0,C 180,E1 25279.764,E2 25279.764} C_VEL
LIN {X 0,Y 84.377,Z 1225.073,A -85,B 0,C 180,E1 25290.004,E2 25290.004} C_VEL
LIN {X 0,Y 87.491,Z 1223.858,A -85,B 0,C 180,E1 25310.183,E2 25310.183} C_VEL
LIN {X 0,Y 102.041,Z 1218.628,A -85,B 0,C 180,E1 25331.253,E2 25331.253} C_VEL
LIN {X 0,Y 128.173,Z 1207.206,A -85,B 0,C 180,E1 25347.834,E2 25347.834} C_VEL
LIN {X 0,Y 156.965,Z 1191.239,A -85,B 0,C 180,E1 25357.719,E2 25357.719} C_VEL
LIN {X 0,Y 171.213,Z 1181.796,A -85,B 0,C 180,E1 25361.185,E2 25361.185} C_VEL
LIN {X 0,Y 176.277,Z 1177.884,A -85,B 0,C 180,E1 25365.12,E2 25365.12} C_VEL
LIN {X 0,Y 182.47,Z 1174.003,A -85,B 0,C 180,E1 25372.94,E2 25372.94} C_VEL
LIN {X 0,Y 187.248,Z 1173.122,A -85,B 0,C 180,E1 25380,E2 25380} C_VEL
LIN {X 0,Y 187.845,Z 1174.048,A -85,B 0,C 180,E1 25382.258,E2 25382.258} C_VEL
LIN {X 0,Y 186.217,Z 1176.837,A -85,B 0,C 180,E1 25384.239,E2 25384.239} C_VEL
LIN {X 0,Y 179.612,Z 1183.316,A -85,B 0,C 180,E1 25386.146,E2 25386.146} C_VEL
LIN {X 0,Y 174.873,Z 1187.337,A -85,B 0,C 180,E1 25386.914,E2 25386.914} C_VEL
LIN {X 0,Y 142.003,Z 1211.342,A -85,B 0,C 180,E1 25393.244,E2 25393.244} C_VEL
LIN {X 0,Y 110.531,Z 1230.153,A -85,B 0,C 180,E1 25404.177,E2 25404.177} C_VEL
LIN {X 0,Y 84.513,Z 1244.089,A -85,B 0,C 180,E1 25424.416,E2 25424.416} C_VEL
LIN {X 0,Y 75.099,Z 1250.491,A -85,B 0,C 180,E1 25446.3,E2 25446.3} C_VEL
LIN {X 0,Y 75.391,Z 1253.268,A -85,B 0,C 180,E1 25469.996,E2 25469.996} C_VEL
LIN {X 0,Y 75.098,Z 1250.516,A -85,B 0,C 180,E1 25493.691,E2 25493.691} C_VEL
LIN {X 0,Y 88.367,Z 1242.052,A -85,B 0,C 180,E1 25520.21,E2 25520.21} C_VEL
LIN {X 0,Y 117.299,Z 1226.452,A -85,B 0,C 180,E1 25538.851,E2 25538.851} C_VEL
LIN {X 0,Y 150.332,Z 1205.837,A -85,B 0,C 180,E1 25548.695,E2 25548.695} C_VEL
LIN {X 0,Y 180.43,Z 1182.897,A -85,B 0,C 180,E1 25553.803,E2 25553.803} C_VEL
LIN {X 0,Y 181.839,Z 1180.71,A -85,B 0,C 180,E1 25555.24,E2 25555.24} C_VEL
LIN {X 0,Y 180.879,Z 1178.308,A -85,B 0,C 180,E1 25560,E2 25560} C_VEL
LIN {X 0,Y 177.687,Z 1178.603,A -85,B 0,C 180,E1 25564.871,E2 25564.871} C_VEL
LIN {X 0,Y 173.791,Z 1180.178,A -85,B 0,C 180,E1 25570,E2 25570} C_VEL
LIN {X 0,Y 167.264,Z 1184.399,A -85,B 0,C 180,E1 25576.508,E2 25576.508} C_VEL
LIN {X 0,Y 136.755,Z 1202.518,A -85,B 0,C 180,E1 25584.453,E2 25584.453} C_VEL
LIN {X 0,Y 108.424,Z 1215.462,A -85,B 0,C 180,E1 25596.849,E2 25596.849} C_VEL
LIN {X 0,Y 88.765,Z 1222.643,A -85,B 0,C 180,E1 25613.491,E2 25613.491} C_VEL
LIN {X 0,Y 77.235,Z 1226.195,A -85,B 0,C 180,E1 25638.737,E2 25638.737} C_VEL
LIN {X 0,Y 76.608,Z 1226.444,A -85,B 0,C 180,E1 25650.004,E2 25650.004} C_VEL
LIN {X 0,Y 80.212,Z 1225.235,A -85,B 0,C 180,E1 25672.106,E2 25672.106} C_VEL
LIN {X 0,Y 95.588,Z 1220.272,A -85,B 0,C 180,E1 25693.705,E2 25693.705} C_VEL
LIN {X 0,Y 122.017,Z 1209.632,A -85,B 0,C 180,E1 25709.968,E2 25709.968} C_VEL
LIN {X 0,Y 153.239,Z 1193.194,A -85,B 0,C 180,E1 25720.19,E2 25720.19} C_VEL
LIN {X 0,Y 167.281,Z 1184.217,A -85,B 0,C 180,E1 25723.594,E2 25723.594} C_VEL
LIN {X 0,Y 170.704,Z 1181.908,A -85,B 0,C 180,E1 25726.513,E2 25726.513} C_VEL
LIN {X 0,Y 173.746,Z 1180.033,A -85,B 0,C 180,E1 25729.997,E2 25729.997} C_VEL
LIN {X 0,Y 178.056,Z 1178.402,A -85,B 0,C 180,E1 25735.895,E2 25735.895} C_VEL
LIN {X 0,Y 181.088,Z 1178.103,A -85,B 0,C 180,E1 25740.242,E2 25740.242} C_VEL
LIN {X 0,Y 181.899,Z 1181.003,A -85,B 0,C 180,E1 25745.418,E2 25745.418} C_VEL
LIN {X 0,Y 178.829,Z 1184.069,A -85,B 0,C 180,E1 25746.375,E2 25746.375} C_VEL
LIN {X 0,Y 174.873,Z 1187.337,A -85,B 0,C 180,E1 25746.914,E2 25746.914} C_VEL
LIN {X 0,Y 160.468,Z 1197.264,A -85,B 0,C 180,E1 25747.671,E2 25747.671} C_VEL
LIN {X 0,Y 145.831,Z 1206.341,A -85,B 0,C 180,E1 25748.796,E2 25748.796} C_VEL
LIN {X 0,Y 111.373,Z 1226.65,A -85,B 0,C 180,E1 25758.47,E2 25758.47} C_VEL
LIN {X 0,Y 81.056,Z 1241.619,A -85,B 0,C 180,E1 25777.694,E2 25777.694} C_VEL
LIN {X 0,Y 67.718,Z 1249.052,A -85,B 0,C 180,E1 25803.528,E2 25803.528} C_VEL
LIN {X 0,Y 67.47,Z 1251.87,A -85,B 0,C 180,E1 25829.995,E2 25829.995} C_VEL
LIN {X 0,Y 67.861,Z 1248.937,A -85,B 0,C 180,E1 25857.197,E2 25857.197} C_VEL
LIN {X 0,Y 85.665,Z 1239.394,A -85,B 0,C 180,E1 25886.789,E2 25886.789} C_VEL
LIN {X 0,Y 114.508,Z 1225.009,A -85,B 0,C 180,E1 25902.724,E2 25902.724} C_VEL
LIN {X 0,Y 146.246,Z 1206.17,A -85,B 0,C 180,E1 25911.31,E2 25911.31} C_VEL
LIN {X 0,Y 173.651,Z 1186.4,A -85,B 0,C 180,E1 25915.673,E2 25915.673} C_VEL
LIN {X 0,Y 175.338,Z 1184.73,A -85,B 0,C 180,E1 25916.423,E2 25916.423} C_VEL
LIN {X 0,Y 174.446,Z 1183.188,A -85,B 0,C 180,E1 25920,E2 25920} C_VEL
LIN {X 0,Y 170.87,Z 1183.502,A -85,B 0,C 180,E1 25925.066,E2 25925.066} C_VEL
LIN {X 0,Y 164.607,Z 1186.283,A -85,B 0,C 180,E1 25932.495,E2 25932.495} C_VEL
LIN {X 0,Y 160.955,Z 1188.548,A -85,B 0,C 180,E1 25934.776,E2 25934.776} C_VEL
LIN {X 0,Y 127.402,Z 1207.019,A -85,B 0,C 180,E1 25943.378,E2 25943.378} C_VEL
LIN {X 0,Y 101.202,Z 1217.858,A -85,B 0,C 180,E1 25954.911,E2 25954.911} C_VEL
LIN {X 0,Y 78.956,Z 1225.022,A -85,B 0,C 180,E1 25975.02,E2 25975.02} C_VEL
LIN {X 0,Y 69.612,Z 1227.57,A -85,B 0,C 180,E1 25997.485,E2 25997.485} C_VEL
LIN {X 0,Y 68.838,Z 1227.815,A -85,B 0,C 180,E1 26010.004,E2 26010.004} C_VEL
LIN {X 0,Y 73.034,Z 1226.614,A -85,B 0,C 180,E1 26034.413,E2 26034.413} C_VEL
LIN {X 0,Y 89.803,Z 1221.74,A -85,B 0,C 180,E1 26056.93,E2 26056.93} C_VEL
LIN {X 0,Y 118.276,Z 1211.022,A -85,B 0,C 180,E1 26073.269,E2 26073.269} C_VEL
LIN {X 0,Y 150.651,Z 1194.646,A -85,B 0,C 180,E1 26082.963,E2 26082.963} C_VEL
LIN {X 0,Y 162.83,Z 1187.17,A -85,B 0,C 180,E1 26085.847,E2 26085.847} C_VEL
LIN {X 0,Y 167.964,Z 1184.414,A -85,B 0,C 180,E1 26091.222,E2 26091.222} C_VEL
LIN {X 0,Y 174.499,Z 1182.988,A -85,B 0,C 180,E1 26100,E2 26100} C_VEL
LIN {X 0,Y 175.397,Z 1184.693,A -85,B 0,C 180,E1 26103.816,E2 26103.816} C_VEL
LIN {X 0,Y 145.831,Z 1206.341,A -85,B 0,C 180,E1 26108.796,E2 26108.796} C_VEL
LIN {X 0,Y 130.762,Z 1214.584,A -85,B 0,C 180,E1 26110.259,E2 26110.259} C_VEL
LIN {X 0,Y 117.157,Z 1220.984,A -85,B 0,C 180,E1 26111.778,E2 26111.778} C_VEL
LIN {X 0,Y 115.401,Z 1221.853,A -85,B 0,C 180,E1 26112.254,E2 26112.254} C_VEL
LIN {X 0,Y 84.202,Z 1236.695,A -85,B 0,C 180,E1 26126.345,E2 26126.345} C_VEL
LIN {X 0,Y 62.683,Z 1246.33,A -85,B 0,C 180,E1 26152.992,E2 26152.992} C_VEL
LIN {X 0,Y 58.404,Z 1249.5,A -85,B 0,C 180,E1 26175.021,E2 26175.021} C_VEL
LIN {X 0,Y 59.529,Z 1250.468,A -85,B 0,C 180,E1 26189.995,E2 26189.995} C_VEL
LIN {X 0,Y 60.487,Z 1247.632,A -85,B 0,C 180,E1 26219.925,E2 26219.925} C_VEL
LIN {X 0,Y 78.762,Z 1239.117,A -85,B 0,C 180,E1 26249.553,E2 26249.553} C_VEL
LIN {X 0,Y 112.143,Z 1223.631,A -85,B 0,C 180,E1 26266.726,E2 26266.726} C_VEL
LIN {X 0,Y 145.505,Z 1204.522,A -85,B 0,C 180,E1 26274.599,E2 26274.599} C_VEL
LIN {X 0,Y 167.055,Z 1189.666,A -85,B 0,C 180,E1 26277.658,E2 26277.658} C_VEL
LIN {X 0,Y 168.58,Z 1188.297,A -85,B 0,C 180,E1 26278.186,E2 26278.186} C_VEL
LIN {X 0,Y 163.969,Z 1188.272,A -85,B 0,C 180,E1 26285.28,E2 26285.28} C_VEL
LIN {X 0,Y 157.867,Z 1190.769,A -85,B 0,C 180,E1 26292.006,E2 26292.006} C_VEL
LIN {X 0,Y 124.168,Z 1208.542,A -85,B 0,C 180,E1 26300.153,E2 26300.153} C_VEL
LIN {X 0,Y 91.363,Z 1221.07,A -85,B 0,C 180,E1 26314.333,E2 26314.333} C_VEL
LIN {X 0,Y 72.684,Z 1226.403,A -85,B 0,C 180,E1 26331.482,E2 26331.482} C_VEL
LIN {X 0,Y 61.624,Z 1229.041,A -85,B 0,C 180,E1 26358.362,E2 26358.362} C_VEL
LIN {X 0,Y 61.624,Z 1229.034,A -85,B 0,C 180,E1 26381.638,E2 26381.638} C_VEL
LIN {X 0,Y 76.756,Z 1225.354,A -85,B 0,C 180,E1 26413.485,E2 26413.485} C_VEL
LIN {X 0,Y 105.778,Z 1216.005,A -85,B 0,C 180,E1 26433.084,E2 26433.084} C_VEL
LIN {X 0,Y 137.748,Z 1201.846,A -85,B 0,C 180,E1 26443.454,E2 26443.454} C_VEL
LIN {X 0,Y 157.908,Z 1190.578,A -85,B 0,C 180,E1 26447.972,E2 26447.972} C_VEL
LIN {X 0,Y 163.911,Z 1188.156,A -85,B 0,C 180,E1 26454.718,E2 26454.718} C_VEL
LIN {X 0,Y 168.64,Z 1188.074,A -85,B 0,C 180,E1 26461.777,E2 26461.777} C_VEL
LIN {X 0,Y 148.733,Z 1202.32,A -85,B 0,C 180,E1 26464.914,E2 26464.914} C_VEL
LIN {X 0,Y 115.401,Z 1221.853,A -85,B 0,C 180,E1 26472.254,E2 26472.254} C_VEL
LIN {X 0,Y 99.927,Z 1228.285,A -85,B 0,C 180,E1 26475.076,E2 26475.076} C_VEL
LIN {X 0,Y 84.525,Z 1233.783,A -85,B 0,C 180,E1 26478.997,E2 26478.997} C_VEL
LIN {X 0,Y 56.34,Z 1244.88,A -85,B 0,C 180,E1 26507.957,E2 26507.957} C_VEL
LIN {X 0,Y 50.641,Z 1248.074,A -85,B 0,C 180,E1 26532.657,E2 26532.657} C_VEL
LIN {X 0,Y 51.583,Z 1249.066,A -85,B 0,C 180,E1 26549.994,E2 26549.994} C_VEL
LIN {X 0,Y 53.538,Z 1246.186,A -85,B 0,C 180,E1 26584.307,E2 26584.307} C_VEL
LIN {X 0,Y 73.647,Z 1238.154,A -85,B 0,C 180,E1 26614.1,E2 26614.1} C_VEL
LIN {X 0,Y 109.634,Z 1222.607,A -85,B 0,C 180,E1 26630.688,E2 26630.688} C_VEL
LIN {X 0,Y 145.903,Z 1202.476,A -85,B 0,C 180,E1 26637.965,E2 26637.965} C_VEL
LIN {X 0,Y 161.034,Z 1192.353,A -85,B 0,C 180,E1 26640,E2 26640} C_VEL
LIN {X 0,Y 156.665,Z 1192.93,A -85,B 0,C 180,E1 26645.527,E2 26645.527} C_VEL
LIN {X 0,Y 153.047,Z 1194.14,A -85,B 0,C 180,E1 26649.618,E2 26649.618} C_VEL
LIN {X 0,Y 132.228,Z 1205.099,A -85,B 0,C 180,E1 26654.07,E2 26654.07} C_VEL
LIN {X 0,Y 99.268,Z 1218.606,A -85,B 0,C 180,E1 26664.212,E2 26664.212} C_VEL
LIN {X 0,Y 71.235,Z 1226.795,A -85,B 0,C 180,E1 26682.154,E2 26682.154} C_VEL
LIN {X 0,Y 54.507,Z 1230.319,A -85,B 0,C 180,E1 26713.934,E2 26713.934} C_VEL
LIN {X 0,Y 53.297,Z 1230.558,A -85,B 0,C 180,E1 26730.006,E2 26730.006} C_VEL
LIN {X 0,Y 59.157,Z 1229.372,A -85,B 0,C 180,E1 26760.681,E2 26760.681} C_VEL
LIN {X 0,Y 81.444,Z 1224.073,A -85,B 0,C 180,E1 26786.233,E2 26786.233} C_VEL
LIN {X 0,Y 112.093,Z 1213.796,A -85,B 0,C 180,E1 26800.459,E2 26800.459} C_VEL
LIN {X 0,Y 146.189,Z 1197.776,A -85,B 0,C 180,E1 26808.698,E2 26808.698} C_VEL
LIN {X 0,Y 153.063,Z 1193.986,A -85,B 0,C 180,E1 26810.371,E2 26810.371} C_VEL
LIN {X 0,Y 158.903,Z 1192.458,A -85,B 0,C 180,E1 26817.565,E2 26817.565} C_VEL
LIN {X 0,Y 161.082,Z 1192.177,A -85,B 0,C 180,E1 26820,E2 26820} C_VEL
LIN {X 0,Y 125.095,Z 1214.539,A -85,B 0,C 180,E1 26825.593,E2 26825.593} C_VEL
LIN {X 0,Y 90.334,Z 1231.291,A -85,B 0,C 180,E1 26836.14,E2 26836.14} C_VEL
LIN {X 0,Y 84.525,Z 1233.783,A -85,B 0,C 180,E1 26838.997,E2 26838.997} C_VEL
LIN {X 0,Y 69.498,Z 1238.286,A -85,B 0,C 180,E1 26844.829,E2 26844.829} C_VEL
LIN {X 0,Y 55.386,Z 1241.744,A -85,B 0,C 180,E1 26853.942,E2 26853.942} C_VEL
LIN {X 0,Y 42.997,Z 1246.648,A -85,B 0,C 180,E1 26889.447,E2 26889.447} C_VEL
LIN {X 0,Y 43.613,Z 1247.66,A -85,B 0,C 180,E1 26909.993,E2 26909.993} C_VEL
LIN {X 0,Y 46.988,Z 1244.738,A -85,B 0,C 180,E1 26949.954,E2 26949.954} C_VEL
LIN {X 0,Y 74.57,Z 1235.158,A -85,B 0,C 180,E1 26982.676,E2 26982.676} C_VEL
LIN {X 0,Y 111.082,Z 1219.948,A -85,B 0,C 180,E1 26995.586,E2 26995.586} C_VEL
LIN {X 0,Y 146.785,Z 1200.431,A -85,B 0,C 180,E1 27001.318,E2 27001.318} C_VEL
LIN {X 0,Y 150.97,Z 1197.815,A -85,B 0,C 180,E1 27001.791,E2 27001.791} C_VEL
LIN {X 0,Y 151.176,Z 1197.026,A -85,B 0,C 180,E1 27003.487,E2 27003.487} C_VEL
LIN {X 0,Y 146.67,Z 1198.321,A -85,B 0,C 180,E1 27007.877,E2 27007.877} C_VEL
LIN {X 0,Y 109.694,Z 1215.3,A -85,B 0,C 180,E1 27015.653,E2 27015.653} C_VEL
LIN {X 0,Y 76.857,Z 1225.672,A -85,B 0,C 180,E1 27029.138,E2 27029.138} C_VEL
LIN {X 0,Y 52.602,Z 1230.782,A -85,B 0,C 180,E1 27054.995,E2 27054.995} C_VEL
LIN {X 0,Y 45.459,Z 1231.885,A -85,B 0,C 180,E1 27095.259,E2 27095.259} C_VEL
LIN {X 0,Y 61.237,Z 1229.113,A -85,B 0,C 180,E1 27137.676,E2 27137.676} C_VEL
LIN {X 0,Y 93.098,Z 1220.901,A -85,B 0,C 180,E1 27158.759,E2 27158.759} C_VEL
LIN {X 0,Y 126.816,Z 1208.018,A -85,B 0,C 180,E1 27168.467,E2 27168.467} C_VEL
LIN {X 0,Y 146.693,Z 1198.146,A -85,B 0,C 180,E1 27172.045,E2 27172.045} C_VEL
LIN {X 0,Y 151.186,Z 1196.887,A -85,B 0,C 180,E1 27176.516,E2 27176.516} C_VEL
LIN {X 0,Y 150.981,Z 1197.67,A -85,B 0,C 180,E1 27178.196,E2 27178.196} C_VEL
LIN {X 0,Y 113.397,Z 1218.724,A -85,B 0,C 180,E1 27183.854,E2 27183.854} C_VEL
LIN {X 0,Y 78.252,Z 1233.758,A -85,B 0,C 180,E1 27195.361,E2 27195.361} C_VEL
LIN {X 0,Y 55.386,Z 1241.744,A -85,B 0,C 180,E1 27213.942,E2 27213.942} C_VEL
LIN {X 0,Y 46.41,Z 1243.803,A -85,B 0,C 180,E1 27224.531,E2 27224.531} C_VEL
LIN {X 0,Y 34.875,Z 1245.496,A -85,B 0,C 180,E1 27251.581,E2 27251.581} C_VEL
LIN {X 0,Y 35.64,Z 1246.253,A -85,B 0,C 180,E1 27269.991,E2 27269.991} C_VEL
LIN {X 0,Y 41.028,Z 1243.288,A -85,B 0,C 180,E1 27317.347,E2 27317.347} C_VEL
LIN {X 0,Y 72.463,Z 1233.715,A -85,B 0,C 180,E1 27348.926,E2 27348.926} C_VEL
LIN {X 0,Y 111.285,Z 1218.225,A -85,B 0,C 180,E1 27360,E2 27360} C_VEL
LIN {X 0,Y 141.472,Z 1202.477,A -85,B 0,C 180,E1 27364.009,E2 27364.009} C_VEL
LIN {X 0,Y 143.111,Z 1201.359,A -85,B 0,C 180,E1 27364.576,E2 27364.576} C_VEL
LIN {X 0,Y 136.588,Z 1204.386,A -85,B 0,C 180,E1 27366.137,E2 27366.137} C_VEL
LIN {X 0,Y 103.271,Z 1218.259,A -85,B 0,C 180,E1 27372.759,E2 27372.759} C_VEL
LIN {X 0,Y 67.774,Z 1228.261,A -85,B 0,C 180,E1 27387.06,E2 27387.06} C_VEL
LIN {X 0,Y 46.416,Z 1232.161,A -85,B 0,C 180,E1 27409.451,E2 27409.451} C_VEL
LIN {X 0,Y 37.746,Z 1233.302,A -85,B 0,C 180,E1 27450.008,E2 27450.008} C_VEL
LIN {X 0,Y 46.409,Z 1232.13,A -85,B 0,C 180,E1 27490.574,E2 27490.574} C_VEL
LIN {X 0,Y 74.722,Z 1226.623,A -85,B 0,C 180,E1 27516.824,E2 27516.824} C_VEL
LIN {X 0,Y 111.394,Z 1215.192,A -85,B 0,C 180,E1 27529.167,E2 27529.167} C_VEL
LIN {X 0,Y 139.923,Z 1202.61,A -85,B 0,C 180,E1 27534.258,E2 27534.258} C_VEL
LIN {X 0,Y 143.085,Z 1201.229,A -85,B 0,C 180,E1 27535.403,E2 27535.403} C_VEL
LIN {X 0,Y 139.53,Z 1203.444,A -85,B 0,C 180,E1 27536.186,E2 27536.186} C_VEL
LIN {X 0,Y 101.916,Z 1222.37,A -85,B 0,C 180,E1 27541.831,E2 27541.831} C_VEL
LIN {X 0,Y 66.088,Z 1235.776,A -85,B 0,C 180,E1 27554.321,E2 27554.321} C_VEL
LIN {X 0,Y 41.042,Z 1243.261,A -85,B 0,C 180,E1 27582.652,E2 27582.652} C_VEL
LIN {X 0,Y 34.875,Z 1245.496,A -85,B 0,C 180,E1 27611.581,E2 27611.581} C_VEL
LIN {X 0,Y 32.237,Z 1245.649,A -85,B 0,C 180,E1 27629.495,E2 27629.495} C_VEL
LIN {X 0,Y 31.384,Z 1242.834,A -85,B 0,C 180,E1 27675.889,E2 27675.889} C_VEL
LIN {X 0,Y 61.064,Z 1235.337,A -85,B 0,C 180,E1 27711.26,E2 27711.26} C_VEL
LIN {X 0,Y 98.153,Z 1222.548,A -85,B 0,C 180,E1 27722.206,E2 27722.206} C_VEL
LIN {X 0,Y 119.27,Z 1213.21,A -85,B 0,C 180,E1 27725.21,E2 27725.21} C_VEL
LIN {X 0,Y 85.063,Z 1224.781,A -85,B 0,C 180,E1 27732.674,E2 27732.674} C_VEL
LIN {X 0,Y 51.968,Z 1231.931,A -85,B 0,C 180,E1 27749.423,E2 27749.423} C_VEL
LIN {X 0,Y 32.688,Z 1234.444,A -85,B 0,C 180,E1 27782.517,E2 27782.517} C_VEL
LIN {X 0,Y 29.954,Z 1234.677,A -85,B 0,C 180,E1 27810.01,E2 27810.01} C_VEL
LIN {X 0,Y 40.788,Z 1233.511,A -85,B 0,C 180,E1 27857.736,E2 27857.736} C_VEL
LIN {X 0,Y 73.099,Z 1227.739,A -85,B 0,C 180,E1 27883.04,E2 27883.04} C_VEL
LIN {X 0,Y 110.577,Z 1216.431,A -85,B 0,C 180,E1 27893.248,E2 27893.248} C_VEL
LIN {X 0,Y 119.492,Z 1212.984,A -85,B 0,C 180,E1 27894.762,E2 27894.762} C_VEL
LIN {X 0,Y 81.283,Z 1228.885,A -85,B 0,C 180,E1 27901.426,E2 27901.426} C_VEL
LIN {X 0,Y 46.242,Z 1239.306,A -85,B 0,C 180,E1 27919.046,E2 27919.046} C_VEL
LIN {X 0,Y 27.054,Z 1244.206,A -85,B 0,C 180,E1 27970.332,E2 27970.332} C_VEL
LIN {X 0,Y 27.656,Z 1244.844,A -85,B 0,C 180,E1 27989.989,E2 27989.989} C_VEL
LIN {X 0,Y 31.384,Z 1242.834,A -85,B 0,C 180,E1 28035.889,E2 28035.889} C_VEL
LIN {X 0,Y 35.36,Z 1241.568,A -85,B 0,C 180,E1 28049.104,E2 28049.104} C_VEL
LIN {X 0,Y 50.167,Z 1236.519,A -85,B 0,C 180,E1 28074.619,E2 28074.619} C_VEL
LIN {X 0,Y 52.096,Z 1236.056,A -85,B 0,C 180,E1 28075.699,E2 28075.699} C_VEL
LIN {X 0,Y 87.29,Z 1225.425,A -85,B 0,C 180,E1 28085.457,E2 28085.457} C_VEL
LIN {X 0,Y 83.691,Z 1226.167,A -85,B 0,C 180,E1 28087.417,E2 28087.417} C_VEL
LIN {X 0,Y 48.601,Z 1233.313,A -85,B 0,C 180,E1 28101.351,E2 28101.351} C_VEL
LIN {X 0,Y 26.021,Z 1235.82,A -85,B 0,C 180,E1 28134.569,E2 28134.569} C_VEL
LIN {X 0,Y 22.182,Z 1236.049,A -85,B 0,C 180,E1 28170.014,E2 28170.014} C_VEL
LIN {X 0,Y 35.999,Z 1234.89,A -85,B 0,C 180,E1 28226.983,E2 28226.983} C_VEL
LIN {X 0,Y 70.234,Z 1229.349,A -85,B 0,C 180,E1 28248.761,E2 28248.761} C_VEL
LIN {X 0,Y 83.721,Z 1226.065,A -85,B 0,C 180,E1 28252.479,E2 28252.479} C_VEL
LIN {X 0,Y 87.315,Z 1225.349,A -85,B 0,C 180,E1 28254.552,E2 28254.552} C_VEL
LIN {X 0,Y 45.708,Z 1237.499,A -85,B 0,C 180,E1 28267.885,E2 28267.885} C_VEL
LIN {X 0,Y 21.919,Z 1242.348,A -85,B 0,C 180,E1 28306.474,E2 28306.474} C_VEL
LIN {X 0,Y 19.653,Z 1243.431,A -85,B 0,C 180,E1 28349.984,E2 28349.984} C_VEL
LIN {X 0,Y 32.236,Z 1240.385,A -85,B 0,C 180,E1 28419.398,E2 28419.398} C_VEL
LIN {X 0,Y 52.096,Z 1236.056,A -85,B 0,C 180,E1 28435.699,E2 28435.699} C_VEL
LIN {X 0,Y 51.997,Z 1235.492,A -85,B 0,C 180,E1 28439.302,E2 28439.302} C_VEL
LIN {X 0,Y 45.648,Z 1235.49,A -85,B 0,C 180,E1 28446.648,E2 28446.648} C_VEL
LIN {X 0,Y 28.319,Z 1236.694,A -85,B 0,C 180,E1 28465.528,E2 28465.528} C_VEL
LIN {X 0,Y 25.872,Z 1236.75,A -85,B 0,C 180,E1 28469.179,E2 28469.179} C_VEL
LIN {X 0,Y 14.417,Z 1237.419,A -85,B 0,C 180,E1 28530.021,E2 28530.021} C_VEL
LIN {X 0,Y 32.412,Z 1236.269,A -85,B 0,C 180,E1 28598.642,E2 28598.642} C_VEL
LIN {X 0,Y 60.807,Z 1232.356,A -85,B 0,C 180,E1 28613.092,E2 28613.092} C_VEL
LIN {X 0,Y 23.291,Z 1239.993,A -85,B 0,C 180,E1 28633.571,E2 28633.571} C_VEL
LIN {X 0,Y 11.624,Z 1242.015,A -85,B 0,C 180,E1 28709.974,E2 28709.974} C_VEL
LIN {X 0,Y 30.334,Z 1238.932,A -85,B 0,C 180,E1 28794.122,E2 28794.122} C_VEL
LIN {X 0,Y 60.445,Z 1232.479,A -85,B 0,C 180,E1 28806.975,E2 28806.975} C_VEL
LIN {X 0,Y 25.872,Z 1236.75,A -85,B 0,C 180,E1 28829.179,E2 28829.179} C_VEL
LIN {X 0,Y 14.702,Z 1237.814,A -85,B 0,C 180,E1 28849.568,E2 28849.568} C_VEL
LIN {X 0,Y 13.389,Z 1238.604,A -85,B 0,C 180,E1 28954.341,E2 28954.341} C_VEL
LIN {X 0,Y 23.732,Z 1238.441,A -85,B 0,C 180,E1 28972.792,E2 28972.792} C_VEL
LIN {X 0,Y 3.593,Z 1240.597,A -85,B 0,C 180,E1 29069.915,E2 29069.915} C_VEL
LIN {X 0,Y 23.703,Z 1238.46,A -85,B 0,C 180,E1 29167.231,E2 29167.231} C_VEL
LIN {X 0,Y 16.088,Z 1238.574,A -85,B 0,C 180,E1 29180.342,E2 29180.342} C_VEL
LIN {X 0,Y 6.642,Z 1238.791,A -85,B 0,C 180,E1 29250.046,E2 29250.046} C_VEL
LIN {X 0,Y 13.389,Z 1238.604,A -85,B 0,C 180,E1 29314.341,E2 29314.341} C_VEL
LIN {X 0,Y 15.188,Z 1240.603,A -85,B 0,C 180,E1 29318.135,E2 29318.135} C_VEL
LIN {X 0,Y 15.188,Z 1319.5,A -85,B 0,C 180,E1 29318.135,E2 29318.135} C_VEL
LIN {X 0,Y 15.188,Z 1319.5,A -85,B 0,C 180,E1 29318.135,E2 29318.135}

